(* PLC project Система умного дома.project, CODESYS CODESYS V3.5 SP17 Patch 3 *)
(* stored: creationDateTime 2026-04-06T20:38:17.5908527, modificationDateTime 2026-03-25T09:46:39.3897592 *)

{attribute 'qualified_only'}
{attribute 'strict'}
TYPE E_ALERT_PRIORITY : (ALERT_PRIORITY_NONE := 0, ALERT_PRIORITY_LOW := 1, ALERT_PRIORITY_MEDIUM := 2, ALERT_PRIORITY_HIGH := 3, ALERT_PRIORITY_CRITICAL := 4) BYTE;
END_TYPE

{attribute 'qualified_only'}
{attribute 'strict'}
TYPE E_Debug_Log_Level : (LOG_LEVEL_MINIMAL := 0, LOG_LEVEL_NORMAL := 1, LOG_LEVEL_VERBOSE := 2, LOG_LEVEL_DEBUG := 3) BYTE;
END_TYPE

{attribute 'qualified_only'}
{attribute 'strict'}
TYPE E_Lifetime_Device_Type : (LIFETIME_DEVICE_PUMP := 1, LIFETIME_DEVICE_FAN := 2) BYTE;
END_TYPE

{attribute 'qualified_only'}
{attribute 'strict'}
TYPE E_Outdoor_Mode : (OUTDOOR_MODE_AUTO := 0, OUTDOOR_MODE_PARTY := 1, OUTDOOR_MODE_SECURITY := 2, OUTDOOR_MODE_ECONOMY := 3, OUTDOOR_MODE_MANUAL := 4) BYTE;
END_TYPE

{attribute 'qualified_only'}
{attribute 'strict'}
TYPE E_PLC_ROLE : (ROLE_UNDEFINED := 0, ROLE_ACTIVE := 1, ROLE_STANDBY := 2, ROLE_OFFLINE := 3) USINT;
END_TYPE

{attribute 'qualified_only'}
{attribute 'strict'}
TYPE E_Rule_Action_Type : (ACTION_NONE := 0, ACTION_SET_FLOOR_HEATING := 1, ACTION_SET_LIGHTING_BASE := 2, ACTION_SET_LIGHTING_ACCENT := 3, ACTION_SET_SOCKET := 4, ACTION_SET_VENTILATION := 5, ACTION_SET_BLINDS := 6, ACTION_ACTIVATE_SCENARIO := 7, ACTION_TOGGLE_LIGHTING := 8, ACTION_TOGGLE_SOCKET := 9) BYTE;
END_TYPE

{attribute 'qualified_only'}
{attribute 'strict'}
TYPE E_Rule_Comparison : (COMP_NONE := 0, COMP_EQ := 1, COMP_GT := 2, COMP_LT := 3, COMP_GE := 4, COMP_LE := 5, COMP_IN_RANGE := 6, COMP_TRUE := 7, COMP_FALSE := 8) BYTE;
END_TYPE

(* values of E_Rule_Condition_Type: COND_AND: Логическое И (Rule Chaining); COND_OR: Логическое ИЛИ (Rule Chaining) *)

{attribute 'qualified_only'}
{attribute 'strict'}
TYPE E_Rule_Condition_Type : (COND_NONE := 0, COND_AIR_TEMP := 1, COND_FLOOR_TEMP := 2, COND_HUMIDITY := 3, COND_CO2 := 4, COND_METHANE := 5, COND_CO := 6, COND_DOOR_WINDOW := 7, COND_FLOOD := 8, COND_SMOKE := 9, COND_MOTION := 10, COND_TIME_OF_DAY := 11, COND_DAY_OF_WEEK := 12, COND_AND := 13, COND_OR := 14) BYTE;
END_TYPE

{attribute 'qualified_only'}
{attribute 'strict'}
TYPE E_SCENARIO_TYPE : (SCENARIO_NONE := 0, SCENARIO_MORNING := 1, SCENARIO_EVENING := 2, SCENARIO_AWAY := 3, SCENARIO_PARTY := 4, SCENARIO_SLEEP := 5, SCENARIO_EMERGENCY := 6, SCENARIO_PRESENCE := 7) BYTE;
END_TYPE

{attribute 'qualified_only'}
{attribute 'strict'}
TYPE E_SENSOR_TYPE : (SENSOR_TYPE_NONE := 0, SENSOR_TYPE_DOOR_WINDOW := 5, SENSOR_TYPE_GLASS_BREAK := 6, SENSOR_TYPE_FLOOD := 7, SENSOR_TYPE_SMOKE := 8, SENSOR_TYPE_GAS_METHANE := 1, SENSOR_TYPE_GAS_CO := 2, SENSOR_TYPE_TEMP_FLOOR := 3, SENSOR_TYPE_TEMP_AIR := 4) USINT;
END_TYPE

{attribute 'qualified_only'}
{attribute 'strict'}
TYPE E_Trend_Parameter_Type : (TREND_PARAM_NONE := 0, TREND_PARAM_TEMP_AIR := 1, TREND_PARAM_TEMP_FLOOR := 2, TREND_PARAM_PRESSURE := 3, TREND_PARAM_PUMP_CURRENT := 4, TREND_PARAM_GAS_METHANE := 5, TREND_PARAM_GAS_CO := 6) BYTE;
END_TYPE

{attribute 'qualified_only'}
{attribute 'strict'}
TYPE E_TwoFactor_Method : (TF_METHOD_NONE := 0, TF_METHOD_RFID := 1, TF_METHOD_TOTP := 2, TF_METHOD_BOTH := 3) BYTE;
END_TYPE

{attribute 'qualified_only'}
{attribute 'strict'}
TYPE E_Valve_Test_Result : (TEST_RESULT_NONE := 0, TEST_RESULT_PASSED := 1, TEST_RESULT_CURRENT_DEVIATION := 2, TEST_RESULT_TIME_DEVIATION := 3, TEST_RESULT_STALL := 4, TEST_RESULT_LIMIT_SWITCH_FAIL := 5, TEST_RESULT_ABORTED := 6) BYTE;
END_TYPE

(* values of E_VALVE_TYPE: VALVE_NC: Нормально-закрытый; VALVE_NO: Нормально-открытый *)

{attribute 'qualified_only'}
{attribute 'strict'}
TYPE E_VALVE_TYPE : (VALVE_NC := 1, VALVE_NO := 2) USINT;
END_TYPE

{attribute 'qualified_only'}
{attribute 'strict'}
TYPE E_VENTILATION_LOCATION : (VENT_LOCATION_NONE := 0, VENT_LOCATION_BASEMENT_GAME_ROOM := 1, VENT_LOCATION_BASEMENT_GYM := 2, VENT_LOCATION_BASEMENT_BOILER_ROOM := 3, VENT_LOCATION_BATHROOM_1F := 4, VENT_LOCATION_BATHROOM_2F := 5, VENT_LOCATION_MASTER_BATHROOM := 6, VENT_LOCATION_LAUNDRY := 7, VENT_LOCATION_KITCHEN := 8) BYTE;
END_TYPE

{attribute 'qualified_only'}
{attribute 'strict'}
TYPE E_VENTILATION_UNIT_TYPE : (VENTILATION_TYPE_NONE := 0, VENTILATION_TYPE_SUPPLY := 1, VENTILATION_TYPE_EXHAUST := 2) USINT;
END_TYPE

{attribute 'qualified_only'}
{attribute 'strict'}
TYPE E_WEATHER_COMPENSATION_METHOD : (WEATHER_COMP_NONE := 0, WEATHER_COMP_OUTDOOR_RESET := 1) USINT;
END_TYPE

{attribute 'qualified_only'}
{attribute 'strict'}
TYPE E_Zone_Access_Level : (ZONE_ACCESS_NONE := 0, ZONE_ACCESS_VIEW := 1, ZONE_ACCESS_CONTROL := 2, ZONE_ACCESS_CONFIG := 3, ZONE_ACCESS_FULL := 4) BYTE;
END_TYPE

TYPE ST_Astro_Time : STRUCT
  sunrise_ms : UDINT := 0;
  sunset_ms : UDINT := 0;
  is_daylight : BOOL := FALSE;
END_STRUCT;
END_TYPE

TYPE ST_BlackBox_Record : STRUCT
  Timestamp : UDINT;
  Gas_Methane_LEL : REAL;
  Gas_CO_PPM : REAL;
  Flood_Active : BOOL;
  Fire_Active : BOOL;
  Valve_Gas_Status : BYTE;
  Valve_Water_Status : BYTE;
  PLC_Active_ID : BYTE;
END_STRUCT;
END_TYPE

TYPE ST_Boiler_Status : STRUCT
  Active : BOOL;
  Running : BOOL;
  Error : BOOL;
  Power_Percent : REAL;
  Current_Power : REAL;
  Work_Seconds : UDINT;
  Work_Hours : REAL;
  Resource_Percent : REAL := 100;
  Last_Start : DT;
END_STRUCT;
END_TYPE

TYPE ST_Component_Maintenance : STRUCT
  Is_Faulty : BOOL;  (* Устройство неисправно *)
  Is_In_Maintenance : BOOL;  (* Выведено в ремонт вручную *)
  Fallback_Value : REAL;  (* Значение для подстановки (0-100% или температура) *)
  Use_Last_Good_Value : BOOL;  (* Использовать последнее достоверное значение *)
END_STRUCT;
END_TYPE

TYPE ST_Debug_Log_Record : STRUCT
  timestamp_ms : UDINT;
  level : BYTE;  (* E_Debug_Log_Level *)
  source_id : BYTE;
  event_code : WORD;
  value_int : UDINT;
  value_real : REAL;
  text : STRING(80);
  crc32 : DWORD;
END_STRUCT;
END_TYPE

TYPE ST_Debug_Logger_Config : STRUCT
  enabled : BOOL;
  sampling_period_ms : UDINT := 1000;
END_STRUCT;
END_TYPE

TYPE ST_Device_Health : STRUCT
  Health_Score : BYTE := 100;  (* 0..100% *)
  Total_Runtime_Hours : UDINT;
  Starts_Count : UDINT;
  Last_Start_Current : REAL;
  Avg_Start_Current : REAL;
  Maintenance_Required : BOOL;
  Warning_Message : STRING(50);
END_STRUCT;
END_TYPE

TYPE ST_DHW_Config : STRUCT
  Target_Temp : REAL := 55;
  Hysteresis : REAL := 2;
  Circulation_Schedule_Enabled : BOOL := TRUE;
  Circulation_Start : TOD := TIME_OF_DAY#6:0;
  Circulation_End : TOD := TIME_OF_DAY#23:0;
  Anti_Legionella_Enabled : BOOL := TRUE;
  Anti_Legionella_Day : UINT := 7;  (* Воскресенье *)
END_STRUCT;
END_TYPE

TYPE ST_DHW_Status : STRUCT
  Temp : REAL;
  Pressure : REAL;
  Heating_Pump_On : BOOL;
  Circ_Pump_On : BOOL;
  Error : BOOL;
  Error_ID : WORD;
END_STRUCT;
END_TYPE

TYPE ST_Flood_Config : STRUCT
  Emergency_Two_Stage_Enabled : BOOL := TRUE;  (* ТЗ 4.4 *)
  Valve_Test_Period_Days : UINT := 7;  (* ТЗ 12.2 *)
  Current_Threshold_MA : REAL := 500;  (* Порог тока для диагностики *)
END_STRUCT;
END_TYPE

TYPE ST_Flood_Global_Config : STRUCT
  valve_types : ARRAY[1..3] OF E_VALVE_TYPE := [3(E_VALVE_TYPE.VALVE_NC)];
  min_duration_ms : UDINT := 30000;
END_STRUCT;
END_TYPE

TYPE ST_FloorHeating_Circuit_Config : STRUCT
  circuit_id : BYTE := 0;
  zone : BYTE := 0;
  design_temp : REAL := 35;
  min_temp : REAL := 20;
  max_temp : REAL := 45;
  pid_kp : REAL := 2;
END_STRUCT;
END_TYPE

TYPE ST_FloorHeating_Global_Config : STRUCT
  enable_floor_heating : BOOL := TRUE;
  anti_freeze_temp : REAL := 7;
  overheat_temp : REAL := 45;
  weather_compensation_enabled : BOOL := TRUE;
  total_circuits : BYTE := 16;
END_STRUCT;
END_TYPE

TYPE ST_FloorHeating_Manifold_Config : STRUCT
  manifold_id : BYTE;
  location : STRING(30);
  nominal_flow : REAL;
  enable_pump : BOOL;
  circuits : ARRAY[1..4] OF ST_FloorHeating_Circuit_Config;
END_STRUCT;
END_TYPE

TYPE ST_Gas_Valve_Configuration : STRUCT
  valve_id : BYTE := 0;
  valve_type : E_VALVE_TYPE := E_VALVE_TYPE.VALVE_NC;
  close_time_seconds : UDINT := 10;
  open_time_seconds : UDINT := 10;
  emergency_open_allowed : BOOL := FALSE;
END_STRUCT;
END_TYPE

TYPE ST_Gateway_Command : STRUCT
  command_id : UDINT;
  timestamp_ms : UDINT;
  operator_id : STRING(10);
  command_type : BYTE;
  target_zone : BYTE;
  target_value : REAL;
  target_on_off : BOOL;
  target_scenario : E_SCENARIO_TYPE;
  target_armed : BOOL;
  crc32 : DWORD;
END_STRUCT;
END_TYPE

TYPE ST_Heating_Config : STRUCT
  Weather_Comp_Enabled : BOOL := TRUE;
  Weather_Coef : REAL := 0.1;
  Freeze_Threshold : REAL := 7;
  Overheat_Threshold : REAL := 45;
  Night_Reduction : REAL := 3;
  Target_Floor_Temp : REAL := 28;
  Target_Room_Temp : REAL := 22;
  Hysteresis : REAL := 0.5;
END_STRUCT;
END_TYPE

TYPE ST_History_Record : STRUCT
  timestamp_ms : UDINT := 0;
  event_code : WORD := 0;
  event_value : REAL := 0;
  unit : BYTE := 0;
  zone_id : BYTE := 0;
  operator_id : STRING(10) := '';
  priority : E_ALERT_PRIORITY := E_ALERT_PRIORITY.ALERT_PRIORITY_NONE;
END_STRUCT;
END_TYPE

TYPE ST_Lifetime_Status : STRUCT
  device_id : BYTE;
  runtime_hours : UDINT;
  start_count : UDINT;
  remaining_hours : UDINT;
  remaining_percent : BYTE;
  maintenance_required : BOOL;
  last_calc_timestamp : UDINT;
END_STRUCT;
END_TYPE

TYPE ST_Maintenance_Access_Config : STRUCT
  maintenance_enabled : BOOL := FALSE;
  max_duration_minutes : UDINT := 60;
  requires_two_person : BOOL := TRUE;
  access_level_required : BYTE := 2;
END_STRUCT;
END_TYPE

TYPE ST_Manifold_Status : STRUCT
  Pump_On : BOOL;
  Pump_Current : REAL;
  Pressure : REAL;
  Temp_Supply : REAL;
  Temp_Return : REAL;
  Valve_Pos : REAL;  (* 0-100% *)
  Error : BOOL;
  Error_ID : WORD;
END_STRUCT;
END_TYPE

TYPE ST_Operator_Zone_Rights : STRUCT
  operator_id : STRING(10);
  global_access_level : BYTE := 0;
  zone_masks : ARRAY[1..18] OF DWORD;
  last_modified : UDINT;
END_STRUCT;
END_TYPE

TYPE ST_Outdoor_Zone_Config : STRUCT
  zone_id : BYTE := 0;
  lighting_circuit_id : BYTE := 0;
  auto_enabled : BOOL := TRUE;
  party_mode_enabled : BOOL := FALSE;
END_STRUCT;
END_TYPE

TYPE ST_Owen_Analog_Value : STRUCT
  rValue : REAL;  (* Измеренное значение *)
  uiCycleTime : UINT;  (* Циклическое время *)
  wStatus : WORD;  (* Код статуса (ANALOG_SENSOR_ERRORS) *)
END_STRUCT;
END_TYPE

TYPE ST_Rule_Action : STRUCT
  Active : BOOL;
  Target_ID : BYTE;
  Value : REAL;
END_STRUCT;
END_TYPE

TYPE ST_Scenario_Config : STRUCT
  scenario_id : E_SCENARIO_TYPE;
  lighting_level_base : BYTE := 100;
  lighting_level_accent : BYTE := 100;
  floor_heating_adjust_celsius : REAL := 0;
  ventilation_speed_percent : BYTE := 50;
  sockets_enabled : BOOL := TRUE;
  blinds_position_percent : BYTE := 0;
END_STRUCT;
END_TYPE

TYPE ST_Scenario_Transition_Config : STRUCT
  current_scenario : E_SCENARIO_TYPE;
  target_scenario : E_SCENARIO_TYPE;
  min_duration_minutes : UDINT := 5;
  transition_allowed : BOOL := FALSE;
END_STRUCT;
END_TYPE

TYPE ST_Security_Config : STRUCT
  PIN_Code : STRING(4) := '1234';
  Max_Attempts : UINT := 3;
  Entry_Delay_S : UINT := 45;
  Two_Factor_Enabled : BOOL := FALSE;
  Two_Stage_Mode : BOOL := TRUE;  (* ТЗ 3.4 *)
  Confirmation_Timeout_S : UINT := 120;  (* ТЗ 3.4 (60-300с) *)
  Phones : ARRAY[1..5] OF STRING(15);
  gate_open_pulse_ms : UDINT := 1000;  (* Управление доступом *)
  wicket_open_pulse_ms : UDINT := 1000;
  lock_open_pulse_ms : UDINT := 1000;
  lock_close_pulse_ms : UDINT := 1000;
END_STRUCT;
END_TYPE

TYPE ST_Security_Global_Config : STRUCT
  entry_delay_seconds : UDINT := 30;
  exit_delay_seconds : UDINT := 60;
  alarm_duration_seconds : UDINT := 180;
  two_person_timeout_seconds : UDINT := 120;
  max_access_attempts : BYTE := 3;
  auto_arm_enabled : BOOL := FALSE;
  auto_arm_time_ms : UDINT := 0;
  gate_open_pulse_ms : UDINT := 1000;  (* ТЗ: Управление доступом *)
  wicket_open_pulse_ms : UDINT := 1000;
  lock_open_pulse_ms : UDINT := 1000;
  lock_close_pulse_ms : UDINT := 1000;
END_STRUCT;
END_TYPE

TYPE ST_Security_Zone_State : STRUCT
  Armed : BOOL;
  Alarm : BOOL;
  Bypassed : BOOL;
  Last_Trigger_Time : DT;
  Trigger_Count : UINT;
END_STRUCT;
END_TYPE

TYPE ST_Sensor_Calibration_Record : STRUCT
  sensor_id : UDINT := 0;
  sensor_type : E_SENSOR_TYPE;
  zone_id : BYTE := 0;
  offset : REAL := 0;
  multiplier : REAL := 1;
  last_calibration_timestamp : UDINT := 0;
  verification_passed : BOOL := FALSE;
END_STRUCT;
END_TYPE

TYPE ST_State_Snapshot : STRUCT
  timestamp_ms : UDINT := 0;
  operator_id : STRING(10) := '';
  scenario_id : E_SCENARIO_TYPE := E_SCENARIO_TYPE.SCENARIO_NONE;
  lighting_levels : ARRAY[1..16] OF BYTE;
  floor_heating_setpoints : ARRAY[1..16] OF REAL;
  alarm_active : BOOL := FALSE;
  crc32 : DWORD := 0;
END_STRUCT;
END_TYPE

TYPE ST_System_State_Summary : STRUCT
  Outdoor_Temp : REAL;
  Indoor_Temp : ARRAY[1..16] OF REAL;
  Floor_Temps : ARRAY[1..16] OF REAL;
  Humidity : ARRAY[1..8] OF REAL;
  CO2 : ARRAY[1..8] OF REAL;
  Gas_Alarm : BOOL;
  Flood_Alarm : BOOL;
  Fire_Alarm : BOOL;
  Security_Armed : BOOL;
END_STRUCT;
END_TYPE

TYPE ST_Tariff_Config : STRUCT
  Enabled : BOOL := FALSE;
  Night_Start_Hour : UINT := 23;  (* 23:00 *)
  Night_End_Hour : UINT := 7;  (* 07:00 *)
  Boost_Delta : REAL := 2;  (* На сколько градусов поднять уставку ночью *)
END_STRUCT;
END_TYPE

TYPE ST_Trend_Config : STRUCT
  param_type : BYTE;  (* E_Trend_Parameter_Type *)
  zone_id : BYTE;
  enabled : BOOL;
  deviation_threshold_percent : REAL := 10;
  history_days : UDINT := 7;
END_STRUCT;
END_TYPE

TYPE ST_Trend_Data : STRUCT
  config : ST_Trend_Config;
  record_count : UDINT;
  write_index : UDINT;
  sum_values : REAL;
  crc32 : DWORD;
END_STRUCT;
END_TYPE

TYPE ST_Trend_Header : STRUCT
  parameter_type : BYTE;  (* E_Trend_Parameter_Type *)
  zone_id : BYTE := 0;
  records_count : UDINT := 0;
  average_value : REAL := 0;
  min_value : REAL := 0;
  max_value : REAL := 0;
END_STRUCT;
END_TYPE

TYPE ST_Trend_History_Record : STRUCT
  timestamp_ms : UDINT := 0;
  value : REAL := 0;
END_STRUCT;
END_TYPE

TYPE ST_TwoFactor_Auth_State : STRUCT
  operator_id : STRING(10);
  is_pending : BOOL;  (* Ожидание ввода 2-го фактора *)
  start_time : UDINT;
  timeout_ms : UDINT := 60000;
END_STRUCT;
END_TYPE

TYPE ST_TwoFactor_Data : STRUCT
  operator_id : STRING(10);
  AuthMethod : BYTE;  (* E_TwoFactor_Method *)
  rfid_tag : STRING(20);
  totp_secret : STRING(32);
  last_modified : UDINT;
END_STRUCT;
END_TYPE

TYPE ST_User_Rule : STRUCT
  Enabled : BOOL;
  Condition_Type : BYTE;  (* 1-Temp, 2-Hum, 3-CO2, 4-Security, 5-Time *)
  Condition_Op : BYTE;  (* 1:>, 2:<, 3:= *)
  Condition_Value : REAL;
  Action_Target_ID : BYTE;
  Action_Value : REAL;
  Action_Type : BYTE;  (* 1-SetTemp, 2-Switch, 3-Scenario *)
  Priority : BYTE;  (* ТЗ 7.4: Приоритет (0-255) *)
END_STRUCT;
END_TYPE

TYPE ST_Valve_Test_Config : STRUCT
  valve_id : BYTE := 0;
  test_interval_days : UDINT := 7;
  nominal_current_a : REAL := 0.5;
  Nominal_Current : REAL := 0.5;
  nominal_close_time_sec : REAL := 10;
  enabled : BOOL := TRUE;
END_STRUCT;
END_TYPE

TYPE ST_Ventilation_Config : STRUCT
  CO2_Threshold : REAL := 800;
  Humidity_Threshold : REAL := 65;
  Night_Mode_Start : TOD := TIME_OF_DAY#23:0;
  Night_Mode_End : TOD := TIME_OF_DAY#7:0;
END_STRUCT;
END_TYPE

TYPE ST_Ventilation_Global_Config : STRUCT
  enable_ventilation : BOOL := TRUE;
  total_units : BYTE := 8;
  default_supply_speed : BYTE := 40;
  default_exhaust_speed : BYTE := 40;
END_STRUCT;
END_TYPE

TYPE ST_Ventilation_Scenario_Mode : STRUCT
  Scenario_ID : BYTE;
  Scenario_Priority : BYTE;
  Fire_Alarm : BOOL;
  Methane_Alarm : BOOL;
  Smoke_Detected : BOOL;
  Exhaust_Modes : ARRAY[1..5] OF BYTE;
  Supply_Modes : ARRAY[1..3] OF BYTE;
END_STRUCT;
END_TYPE

TYPE ST_Ventilation_Unit : STRUCT
  Enabled : BOOL;
  Speed_Percent : REAL;
  Filter_Dirty : BOOL;
  Error : BOOL;
  Mode : BYTE;  (* 0-Eco, 1-Std, 2-Int, 3-Emergency *)
END_STRUCT;
END_TYPE

TYPE ST_Ventilation_Unit_Config : STRUCT
  unit_id : BYTE := 0;
  unit_type : E_VENTILATION_UNIT_TYPE;
  location : E_VENTILATION_LOCATION;
  min_speed : BYTE := 20;
  max_speed : BYTE := 100;
  Threshold_Hum : REAL := 65;
  has_smoke_detector : BOOL := FALSE;
END_STRUCT;
END_TYPE

TYPE ST_Zone_Sensors : STRUCT
  Temp_Room : REAL;
  Temp_Floor : REAL;
  Motion_Active : BOOL;
  Switch_Physical : BOOL;
  Light_State : BOOL;
  Maintenance : ST_Component_Maintenance;
END_STRUCT;
END_TYPE

{attribute 'qualified_only'}
VAR_GLOBAL  (* GVL_BlackBox *)
  G_BlackBox_Buffer : ARRAY[0..99] OF ST_BlackBox_Record;  (* Буфер на 100 записей (при опросе 100мс это 10 секунд истории) *)
  G_BlackBox_Frozen : BOOL;
  G_BlackBox_LastIndex : INT;
END_VAR

{attribute 'qualified_only'}
VAR_GLOBAL CONSTANT  (* GVL_Constants *)
  C_MS_PER_SEC : UDINT := 1000;
  C_SEC_PER_MIN : UDINT := 60;
  C_MIN_PER_HOUR : UDINT := 60;
  C_MS_PER_MIN : UDINT := 60000;
  C_MAX_RULES : INT := 20;
  C_ZONE_COUNT : BYTE := 18;
END_VAR

{attribute 'qualified_only'}
VAR_GLOBAL  (* GVL_Diagnostics *)
  G_Pump_Health : ARRAY[1..5] OF ST_Device_Health;  (* Для 5 коллекторных насосов *)
  G_Gas_Valve_Health : ST_Device_Health;
  G_System_Health_Summary : BYTE := 100;
END_VAR

{attribute 'qualified_only'}
VAR_GLOBAL  (* GVL_Global_Variables *)
  GVL_System_Time_MS : UDINT;
  GVL_IsActivePLC : BOOL := TRUE;
  GVL_Local_PLC_Role : E_PLC_ROLE := E_PLC_ROLE.ROLE_ACTIVE;
  GVL_Floor_Temps : ARRAY[1..16] OF REAL;  (* Данные датчиков *)
  GVL_Valve_States : ARRAY[1..3] OF BYTE;
END_VAR

VAR_GLOBAL  (* GVL_HMI_Config *)
  G_HMI_FloorHeating_Configs : ARRAY[1..16] OF ST_FloorHeating_Circuit_Config;  (* Настройки отопления (16 контуров) *)
  G_HMI_Tariff_Settings : ST_Tariff_Config;
  G_HMI_Vent_Global_Config : ST_Ventilation_Global_Config;  (* Настройки вентиляции (8 установок) *)
  G_HMI_Vent_Unit_Configs : ARRAY[1..8] OF ST_Ventilation_Unit_Config;
  G_HMI_Scenario_Configs : ARRAY[1..6] OF ST_Scenario_Config;  (* Для каждого типа сценария *)
  G_HMI_Outdoor_Configs : ARRAY[1..4] OF ST_Outdoor_Zone_Config;
  G_HMI_Flood_Config : ST_Flood_Global_Config;  (* Настройки безопасности *)
  G_HMI_Cleaning_Mode_Active : ARRAY[1..3] OF BOOL;  (* Режим уборки для 3-х зон протечки *)
  G_HMI_Cleaning_Mode_TimeLeft : ARRAY[1..3] OF UINT;  (* Оставшееся время (мин) *)
  G_HMI_Gas_Config : ST_Gas_Valve_Configuration;
  G_HMI_Admin_2FA_Enabled : BOOL := FALSE;  (* Настройка: 1 или 2 фактора для ADMIN *)
  G_HMI_Current_Operator_Factor2_Done : BOOL;  (* Флаг прохождения 2-го фактора *)
  G_HMI_Sensor_Calibrations : ARRAY[1..20] OF ST_Sensor_Calibration_Record;  (* Калибровка датчиков (например, для 20 датчиков) *)
  G_HMI_Current_Operator_ID : STRING(10);  (* ID текущего авторизованного пользователя *)
  G_HMI_Manual_Gas_Valve_Open : BOOL;  (* Запрос на открытие *)
  G_HMI_Manual_Gas_Valve_Time : UDINT := 5;  (* Время в минутах *)
  G_HMI_Manual_Gas_Valve_TimeLeft : UDINT;  (* Оставшееся время (для вывода на HMI) *)
  G_HMI_Apply_Settings : BOOL;  (* Команда на сохранение настроек в NVRAM *)
  G_HMI_Gate_Open_Req : BOOL;  (* Управление доступом (HMI) *)
  G_HMI_Wicket_Open_Req : BOOL;
  G_HMI_Lock_1_Open_Req : BOOL;
  G_HMI_Lock_1_Close_Req : BOOL;
  G_HMI_Lock_2_Open_Req : BOOL;
  G_HMI_Lock_2_Close_Req : BOOL;
END_VAR

VAR_GLOBAL  (* GVL_IO *)
  DI_Security_Open : ARRAY[1..15] OF BOOL;  (* Датчики открытия (15 физических каналов по ТЗ 3.1) *)
  DI_Security_Glass : ARRAY[1..15] OF BOOL;  (* Датчики разбития (15 физических каналов по ТЗ 3.2) *)
  DI_Security_2F_Group : BOOL;  (* Групповой канал 2-го этажа *)
  DI_Flood_Sensors : ARRAY[1..12] OF BOOL;  (* Датчики протечки (12 штук по ТЗ 4.1) *)
  AO_Manifold_Valves : ARRAY[1..5] OF UINT;  (* 0-1000 (Modbus) *)
  DO_Manifold_Pumps : ARRAY[1..5] OF BOOL;
  AI_Manifold_Currents : ARRAY[1..5] OF INT;  (* 4-20mA -> 400-2000 *)
  AI_Manifold_Pressures : ARRAY[1..5] OF INT;  (* 0-10V -> 0-1000 *)
  AI_Manifold_Temps_Supply : ARRAY[1..5] OF ST_Owen_Analog_Value;
  AI_Manifold_Temps_Return : ARRAY[1..5] OF INT;
  AO_Supply_Fans : ARRAY[1..3] OF UINT;  (* 0-1000 *)
  AO_Exhaust_Fans : ARRAY[1..5] OF UINT;  (* 0-1000 *)
  DO_Boiler_Enable : ARRAY[1..2] OF BOOL;  (* Котлы (BAXI Luna Platinum+ через OpenTherm) *)
  AO_Boiler_Setpoint : ARRAY[1..2] OF UINT;  (* 0-1000 (0-100.0 C) *)
  AI_Boiler_Modulation : ARRAY[1..2] OF INT;
  AI_Boiler_Flame_Status : ARRAY[1..2] OF BOOL;
  DI_Boiler_Error : ARRAY[1..2] OF BOOL;
  AI_Methane_LEL : ARRAY[1..2] OF ST_Owen_Analog_Value;  (* 0-100% LEL *)
  AI_CO_PPM : ARRAY[1..8] OF REAL;  (* 0-1000 PPM *)
  DI_Smoke_Sensors : ARRAY[1..6] OF BOOL;
  AI_Temp_Outdoor : ST_Owen_Analog_Value;  (* Аналоговые входы (AI) *)
  AI_Floor_Temps : ARRAY[1..16] OF REAL;
  AI_Room_Temps : ARRAY[1..16] OF REAL;  (* Датчики температуры помещения (ТЗ 1.1) *)
  DO_Zone_Valves : ARRAY[1..16] OF BOOL;  (* Клапаны контуров ТП *)
  AI_DHW_Temp : REAL;  (* ГВС (ТЗ 5.0) *)
  AI_DHW_Pressure : REAL;
  DO_DHW_Heating_Pump : BOOL;
  DO_DHW_Circ_Pump : BOOL;
  DI_Lighting_Switches : ARRAY[1..16] OF BOOL;  (* Освещение и Движение (ТЗ 1.0, 2.0) *)
  DI_Motion_Sensors : ARRAY[1..16] OF BOOL;
  DO_Gas_Valve_Close : BOOL;  (* Безопасность и Аварии *)
  DO_Water_Valve_35_Close : BOOL;
  DO_Water_Valve_36_Close : BOOL;
  AI_Water_Valve_35_Current : REAL;
  AI_Water_Valve_36_Current : REAL;
  DI_Power_OK : BOOL;
  DO_Gas_Siren : BOOL;
  DO_Fire_Siren : BOOL;
  DO_Pump_Main_Enable : BOOL;
  DO_Gate_Open : BOOL;  (* Управление доступом (Сухие контакты) *)
  DO_Wicket_Open : BOOL;
  DO_Lock_1_Open : BOOL;
  DO_Lock_1_Close : BOOL;
  DO_Lock_2_Open : BOOL;
  DO_Lock_2_Close : BOOL;
END_VAR

VAR_GLOBAL  (* GVL_Vars *)
  G_System_Time_MS : UDINT;  (* Системное время (мс) *)
  G_Current_Scenario : E_SCENARIO_TYPE := E_SCENARIO_TYPE.SCENARIO_NONE;
  G_Security_Armed : BOOL := FALSE;
  G_Gas_Alarm_Active : BOOL := FALSE;
  G_Fire_Alarm_Active : BOOL := FALSE;
  G_Flood_Alarm_Active : BOOL := FALSE;
  G_Local_PLC_ID : BYTE := 1;  (* ID текущего ПЛК (1 для A, 2 для B) *)
  G_Active_PLC_ID : BYTE := 1;  (* ID активного ПЛК в данный момент *)
  G_Remote_PLC_Pulse : BOOL;  (* Импульс от партнера *)
  G_HMI_Current_Operator_ID : STRING(10) := 'ADMIN';  (* HMI и Конфигурация *)
  G_HMI_Gas_Config : ST_Gas_Valve_Configuration;
  G_Heating_Config : ST_Heating_Config;
  G_Ventilation_Config : ST_Ventilation_Config;
  G_DHW_Config : ST_DHW_Config;
  G_Security_Config : ST_Security_Config;
  G_Flood_Config : ST_Flood_Config;
  G_HMI_Mute_Alarm : BOOL;
  G_HMI_Manual_Gas_Valve_Open : BOOL;
  G_HMI_Manual_Gas_Valve_Time : UDINT := 300000;  (* 5 минут по умолчанию *)
  G_HMI_Manual_Gas_Valve_TimeLeft : UDINT;
  G_Floor_Temps : ARRAY[1..16] OF REAL;  (* Состояние датчиков *)
  G_BlackBox_Buffer : ARRAY[0..99] OF ST_BlackBox_Record;  (* Черный ящик *)
  G_BlackBox_LastIndex : INT;
  G_BlackBox_Frozen : BOOL;
  G_Maintenance_Zones : ARRAY[1..16] OF ST_Component_Maintenance;  (* ТЗ 6.0: Обслуживание и ремонт *)
  G_Maintenance_Manifolds : ARRAY[1..5] OF ST_Component_Maintenance;
  G_Maintenance_Lighting : ARRAY[1..16] OF ST_Component_Maintenance;
  G_HMI_Gate_Open_Req : BOOL;  (* Управление доступом (HMI) *)
  G_HMI_Wicket_Open_Req : BOOL;
  G_HMI_Lock_1_Open_Req : BOOL;
  G_HMI_Lock_1_Close_Req : BOOL;
  G_HMI_Lock_2_Open_Req : BOOL;
  G_HMI_Lock_2_Close_Req : BOOL;
END_VAR

INTERFACE IValveController
METHOD OpenValve : BOOL
  VAR_INPUT
    VI_Operator_ID : STRING(10);
    VI_Force : BOOL;
  END_VAR
END_METHOD
METHOD CloseValve : BOOL
  VAR_INPUT
    VI_Operator_ID : STRING(10);
    VI_Force : BOOL;
  END_VAR
END_METHOD
METHOD GetStatus : BYTE
END_METHOD
END_INTERFACE

FUNCTION_BLOCK FB_AccessCode_Manager
  VAR_INPUT
    VI_System_Time_MS : UDINT;
    VI_IsActivePLC : BOOL;
    VI_Code_To_Check : STRING(4);
    VI_RFID_To_Check : STRING(20);
  END_VAR
  VAR_OUTPUT
    VO_Code_Valid : BOOL;
  END_VAR
  VAR_IN_OUT
    VI_Access_Codes : ARRAY[1..GVL_CONSTANTS.C_MAX_ACCESS_CODES] OF DWORD;
    VI_RFID_Tags : ARRAY[1..GVL_CONSTANTS.C_MAX_ACCESS_CODES] OF STRING(20);
  END_VAR
  VAR
    L_i : INT;
    pCode : POINTER TO BYTE;
    L_CRC_Calc : FB_CRC32_Calculator;
    L_Input_Hash : DWORD;
  END_VAR

            VO_Code_Valid := FALSE;

// Вычисляем хэш введенного кода
IF LEN(VI_Code_To_Check) > 0 THEN
    pCode := ADR(VI_Code_To_Check);
    L_Input_Hash := 0;
    FOR L_i := 1 TO GVL_CONSTANTS.C_MAX_ACCESS_CODES DO
        IF VI_Access_Codes[L_i] <> 0 AND VI_Access_Codes[L_i] = L_Input_Hash THEN
            VO_Code_Valid := TRUE;
            RETURN;
        END_IF;
    END_FOR;
END_IF;

// Проверяем RFID метку
IF LEN(VI_RFID_To_Check) > 0 THEN
    FOR L_i := 1 TO GVL_CONSTANTS.C_MAX_ACCESS_CODES DO
        IF VI_RFID_Tags[L_i] <> '' AND VI_RFID_Tags[L_i] = VI_RFID_To_Check THEN
            VO_Code_Valid := TRUE;
            RETURN;
        END_IF;
    END_FOR;
END_IF;
// >>> BULK_SYNC_ANCHOR: FB_AccessCode_Manager <<<
          
END_FUNCTION_BLOCK

FUNCTION_BLOCK FB_Access_Control
  VAR_INPUT
    VI_System_Time_MS : UDINT;
    VI_IsActivePLC : BOOL;
    VI_Armed : BOOL;
    VI_System_Mode : E_System_Operating_Mode;
    VI_Gate_Open_Req : BOOL;
    VI_Wicket_Open_Req : BOOL;
    VI_Lock_1_Open_Req : BOOL;
    VI_Lock_1_Close_Req : BOOL;
    VI_Lock_2_Open_Req : BOOL;
    VI_Lock_2_Close_Req : BOOL;
    VI_PIN_Code : STRING(4);
    VI_RFID_Tag : STRING(20);
    VI_Config : ST_Security_Global_Config;
  END_VAR
  VAR_OUTPUT
    VO_Gate_Open : BOOL;
    VO_Wicket_Open : BOOL;
    VO_Lock_1_Open : BOOL;
    VO_Lock_1_Close : BOOL;
    VO_Lock_2_Open : BOOL;
    VO_Lock_2_Close : BOOL;
  END_VAR
  VAR_IN_OUT
    VI_Access_Codes : ARRAY[1..GVL_CONSTANTS.C_MAX_ACCESS_CODES] OF DWORD;
    VI_RFID_Tags : ARRAY[1..GVL_CONSTANTS.C_MAX_ACCESS_CODES] OF STRING(20);
  END_VAR
  VAR
    L_Gate_Timer : TP;
    L_Wicket_Timer : TP;
    L_Lock_1_Open_T : TP;
    L_Lock_1_Close_T : TP;
    L_Lock_2_Open_T : TP;
    L_Lock_2_Close_T : TP;
    L_Prev_Armed : BOOL;
    L_Auto_Lock_Req : BOOL;
    R_Trig_Gate : R_TRIG;
    R_Trig_Wicket : R_TRIG;
    R_Trig_Lock_1_O : R_TRIG;
    R_Trig_Lock_1_C : R_TRIG;
    R_Trig_Lock_2_O : R_TRIG;
    R_Trig_Lock_2_C : R_TRIG;
    fbAccessCode : FB_AccessCode_Manager;
    L_Valid_PIN : BOOL;
  END_VAR

            // Если ПЛК находится в режиме Standby (резерв), он не должен управлять выходами
IF NOT VI_IsActivePLC THEN
    RETURN;
END_IF;

IF VI_System_Mode = E_System_Operating_Mode.MODE_SAFE_STOP THEN
    VO_Gate_Open := FALSE;
    VO_Wicket_Open := FALSE;
    VO_Lock_1_Open := FALSE;
    VO_Lock_2_Open := FALSE;
    RETURN;
END_IF;

// 1. Логика автоматического закрытия замков при постановке на охрану (ТЗ 3.0)
// При переходе системы в режим "Охрана" принудительно блокируем все замки
IF VI_Armed AND NOT L_Prev_Armed THEN
    L_Auto_Lock_Req := TRUE;
END_IF;
L_Prev_Armed := VI_Armed;

// Детекторы фронта для команд
R_Trig_Gate(CLK := VI_Gate_Open_Req);
R_Trig_Wicket(CLK := VI_Wicket_Open_Req);
R_Trig_Lock_1_O(CLK := VI_Lock_1_Open_Req);
R_Trig_Lock_1_C(CLK := VI_Lock_1_Close_Req OR L_Auto_Lock_Req);
R_Trig_Lock_2_O(CLK := VI_Lock_2_Open_Req);
R_Trig_Lock_2_C(CLK := VI_Lock_2_Close_Req OR L_Auto_Lock_Req);

// Проверка PIN-кода или RFID-метки через менеджер кодов
fbAccessCode(
    VI_System_Time_MS := VI_System_Time_MS,
    VI_IsActivePLC := VI_IsActivePLC,
    VI_Code_To_Check := VI_PIN_Code,
    VI_RFID_To_Check := VI_RFID_Tag,
    VI_Access_Codes := VI_Access_Codes,
    VI_RFID_Tags := VI_RFID_Tags,
    VO_Code_Valid => L_Valid_PIN
);

// 2. Формирование импульсов управления исполнительными механизмами (Pulse Control)
// Открытие ворот и калитки требует валидного ПИН-кода или RFID-метки, если система под охраной
L_Gate_Timer(IN := R_Trig_Gate.Q AND (NOT VI_Armed OR L_Valid_PIN), PT := TO_TIME(VI_Config.gate_open_pulse_ms));
VO_Gate_Open := L_Gate_Timer.Q;

L_Wicket_Timer(IN := R_Trig_Wicket.Q AND (NOT VI_Armed OR L_Valid_PIN), PT := TO_TIME(VI_Config.wicket_open_pulse_ms));
VO_Wicket_Open := L_Wicket_Timer.Q;

L_Lock_1_Open_T(IN := R_Trig_Lock_1_O.Q AND (NOT VI_Armed OR L_Valid_PIN), PT := TO_TIME(VI_Config.lock_open_pulse_ms));
VO_Lock_1_Open := L_Lock_1_Open_T.Q;

L_Lock_1_Close_T(IN := R_Trig_Lock_1_C.Q, PT := TO_TIME(VI_Config.lock_close_pulse_ms));
VO_Lock_1_Close := L_Lock_1_Close_T.Q;

L_Lock_2_Open_T(IN := R_Trig_Lock_2_O.Q AND (NOT VI_Armed OR L_Valid_PIN), PT := TO_TIME(VI_Config.lock_open_pulse_ms));
VO_Lock_2_Open := L_Lock_2_Open_T.Q;

L_Lock_2_Close_T(IN := R_Trig_Lock_2_C.Q, PT := TO_TIME(VI_Config.lock_close_pulse_ms));
VO_Lock_2_Close := L_Lock_2_Close_T.Q;

// Сброс флага автоматического закрытия
IF L_Auto_Lock_Req THEN
    L_Auto_Lock_Req := FALSE;
END_IF;
// >>> BULK_SYNC_ANCHOR: FB_Access_Control <<<
          
END_FUNCTION_BLOCK

FUNCTION_BLOCK FB_Alarm_Compatibility_Package
  VAR_INPUT
    VI_Alarm_Legacy : ST_Alarm_Record;
  END_VAR
  VAR_OUTPUT
    VO_OK : BOOL;
    VO_Alarm_Legacy_Roundtrip : ST_Alarm_Record;
  END_VAR

            VO_OK := TRUE;
VO_Alarm_Legacy_Roundtrip := VI_Alarm_Legacy;
          
END_FUNCTION_BLOCK

FUNCTION_BLOCK FB_Alarm_Manager
  VAR_INPUT
    VI_System_Time_MS : UDINT;
    VI_IsActivePLC : BOOL;
    VI_Gas_Alarm : BOOL;
    VI_Fire_Alarm : BOOL;
    VI_Flood_Alarm : BOOL;
    VI_Security_Alarm : BOOL;
    VI_First_Fault_Active : BOOL;
    VI_First_Fault_Type : INT;
    VI_First_Fault_Source : INT;
    VI_Security_Msg : STRING(200);
    VI_Acknowledge_All : BOOL;
    VI_Mute_Siren : BOOL;
  END_VAR
  VAR_OUTPUT
    VO_Global_Critical : BOOL;
    VO_Global_Warning : BOOL;
    VO_Siren_Active : BOOL;
    VO_Active_Count : INT;
    VO_Unacked_Count : INT;
    VO_Event_Pulse : BOOL;
    VO_Event_Code : UDINT;
    VO_Event_Value : REAL;
    VO_Alarm_List : ARRAY[1..GVL_CONSTANTS.C_MAX_ALARMS] OF ST_Alarm_Record;
  END_VAR
  VAR_IN_OUT
    VI_Boiler_Errors : ARRAY[1..GVL_CONSTANTS.C_MAX_BOILERS] OF BOOL;
  END_VAR
  VAR_IN_OUT
    VIO_Next_Alarm_ID : UDINT;
  END_VAR
  VAR
    fbCompatAlarm : ARRAY[1..GVL_CONSTANTS.C_MAX_ALARMS] OF FB_Alarm_Compatibility_Package;
    L_i, L_j, L_k : INT;
    L_Target_Slot : INT;
    L_Min_Pri : INT;
    L_Pending_Alarms : ARRAY[1..10] OF ST_Alarm_Record;
    L_Pending_Count : INT := 0;
    T_Debounce_Gas : FB_System_Timer;
    T_Debounce_Fire : FB_System_Timer;
    T_Debounce_Flood : FB_System_Timer;
    T_Debounce_Security : FB_System_Timer;
    R_Trig_Gas : R_TRIG;
    R_Trig_Fire : R_TRIG;
    R_Trig_Flood : R_TRIG;
    R_Trig_Security : R_TRIG;
    R_Trig_First_Fault : R_TRIG;
    R_Trig_Boiler : ARRAY[1..GVL_CONSTANTS.C_MAX_BOILERS] OF R_TRIG;
    L_First_Fault_Source_Text : STRING(32);
    L_First_Fault_Type_Text : STRING(32);
    L_Event_Pulse_Latched : BOOL;
    L_Alarm_Compat_All_OK : BOOL;
    L_Alarm_First_Warning : STRING(255);
    L_Alarm_First_Warning_Latched : BOOL;
    L_Alarm_Shadow_Mismatch : BOOL;
    L_Alarm_Shadow_First_Mismatch : INT;
    L_Alarm_V2_Switch_Enabled : BOOL;
    L_Alarm_V2_Path_Ready : BOOL;
    L_Alarm_Using_Legacy_Fallback : BOOL;
    fbAlarmV2Core : FB_Alarm_V2_Core;
    fbHistoryV2Core : FB_History_V2_Core;
    fbBlackBoxV2Core : FB_BlackBox_V2_Core;
    L_BlackBox_V2_Snapshot_Shadow : ST_BlackBox_Snapshot_V2;
    L_History_V2_Shadow_Diff_Found : BOOL;
    L_History_V2_Shadow_First_Diff_Slot : INT;
    L_BlackBox_V2_Shadow_Diff_Found : BOOL;
    L_History_V2_Buffer_Shadow : ARRAY[1..GVL_CONSTANTS.C_MAX_HISTORY_RECORDS] OF ST_History_Event_V2;
    L_Alarm_V2_Shadow_Compare_Enabled : BOOL;
    L_Alarm_V2_Shadow_Diff_Found : BOOL;
    L_Alarm_V2_Shadow_First_Diff_Slot : INT;
    L_Alarm_V2_Event_Pulse : BOOL;
    L_Alarm_V2_Event_Code : UDINT;
    L_Alarm_V2_Event_Value : REAL;
    L_Alarm_V2_List_Shadow : ARRAY[1..GVL_CONSTANTS.C_MAX_ALARMS] OF ST_Alarm_Record;
    L_Alarm_V2_Next_ID_Shadow : UDINT;
  END_VAR

            VO_Event_Pulse := FALSE;
VO_Event_Code := 0;
VO_Event_Value := 0.0;

L_Alarm_Compat_All_OK := TRUE;
L_Alarm_First_Warning := '';
L_Alarm_First_Warning_Latched := FALSE;
L_Alarm_Shadow_Mismatch := FALSE;
L_Alarm_Shadow_First_Mismatch := 0;
L_Alarm_V2_Switch_Enabled := TRUE;
L_Alarm_V2_Path_Ready := FALSE;
L_Alarm_Using_Legacy_Fallback := TRUE;
L_Alarm_V2_Shadow_Compare_Enabled := TRUE;
L_Alarm_V2_Shadow_Diff_Found := FALSE;
L_Alarm_V2_Shadow_First_Diff_Slot := 0;
L_Alarm_V2_Event_Pulse := FALSE;
L_Alarm_V2_Event_Code := 0;
L_Alarm_V2_Event_Value := 0.0;
L_Alarm_V2_Next_ID_Shadow := VIO_Next_Alarm_ID;
L_History_V2_Shadow_Diff_Found := FALSE;
L_History_V2_Shadow_First_Diff_Slot := 0;
L_BlackBox_V2_Shadow_Diff_Found := FALSE;

// 1. Детекция новых тревог (антидребезг + передний фронт)
T_Debounce_Gas(IN := VI_Gas_Alarm, PT := T#100ms, VI_System_Time_MS := VI_System_Time_MS);
T_Debounce_Fire(IN := VI_Fire_Alarm, PT := T#100ms, VI_System_Time_MS := VI_System_Time_MS);
T_Debounce_Flood(IN := VI_Flood_Alarm, PT := T#500ms, VI_System_Time_MS := VI_System_Time_MS);
T_Debounce_Security(IN := VI_Security_Alarm, PT := T#100ms, VI_System_Time_MS := VI_System_Time_MS);

R_Trig_Gas(CLK := T_Debounce_Gas.Q);
R_Trig_Fire(CLK := T_Debounce_Fire.Q);
R_Trig_Flood(CLK := T_Debounce_Flood.Q);
R_Trig_Security(CLK := T_Debounce_Security.Q);
R_Trig_First_Fault(CLK := VI_First_Fault_Active);
FOR L_i := 1 TO GVL_CONSTANTS.C_MAX_BOILERS DO
    R_Trig_Boiler[L_i](CLK := VI_Boiler_Errors[L_i]);
END_FOR;

// 2. Добавление новых тревог в список (Кольцевой буфер)
L_Pending_Count := 0;
L_Event_Pulse_Latched := FALSE;

IF R_Trig_Gas.Q AND L_Pending_Count < 10 THEN
    L_Pending_Count := L_Pending_Count + 1;
    L_Pending_Alarms[L_Pending_Count].Timestamp_MS := VI_System_Time_MS;
    L_Pending_Alarms[L_Pending_Count].Source := 'Gas';
    L_Pending_Alarms[L_Pending_Count].Source_ID := 0;
    L_Pending_Alarms[L_Pending_Count].Message := 'Критическая концентрация газа!';
    L_Pending_Alarms[L_Pending_Count].Severity := E_ALERT_PRIORITY.ALERT_PRIORITY_CRITICAL;
    L_Pending_Alarms[L_Pending_Count].Is_Active := TRUE;
    L_Pending_Alarms[L_Pending_Count].Is_Acknowledged := FALSE;
END_IF;

IF R_Trig_Fire.Q AND L_Pending_Count < 10 THEN
    L_Pending_Count := L_Pending_Count + 1;
    L_Pending_Alarms[L_Pending_Count].Timestamp_MS := VI_System_Time_MS;
    L_Pending_Alarms[L_Pending_Count].Source := 'Fire';
    L_Pending_Alarms[L_Pending_Count].Source_ID := 0;
    L_Pending_Alarms[L_Pending_Count].Message := 'Обнаружено задымление!';
    L_Pending_Alarms[L_Pending_Count].Severity := E_ALERT_PRIORITY.ALERT_PRIORITY_CRITICAL;
    L_Pending_Alarms[L_Pending_Count].Is_Active := TRUE;
    L_Pending_Alarms[L_Pending_Count].Is_Acknowledged := FALSE;
END_IF;

IF R_Trig_Flood.Q AND L_Pending_Count < 10 THEN
    L_Pending_Count := L_Pending_Count + 1;
    L_Pending_Alarms[L_Pending_Count].Timestamp_MS := VI_System_Time_MS;
    L_Pending_Alarms[L_Pending_Count].Source := 'Flood';
    L_Pending_Alarms[L_Pending_Count].Source_ID := 0;
    L_Pending_Alarms[L_Pending_Count].Message := 'Обнаружена протечка воды!';
    L_Pending_Alarms[L_Pending_Count].Severity := E_ALERT_PRIORITY.ALERT_PRIORITY_CRITICAL;
    L_Pending_Alarms[L_Pending_Count].Is_Active := TRUE;
    L_Pending_Alarms[L_Pending_Count].Is_Acknowledged := FALSE;
END_IF;

IF R_Trig_Security.Q AND L_Pending_Count < 10 THEN
    L_Pending_Count := L_Pending_Count + 1;
    L_Pending_Alarms[L_Pending_Count].Timestamp_MS := VI_System_Time_MS;
    L_Pending_Alarms[L_Pending_Count].Source := 'Security';
    L_Pending_Alarms[L_Pending_Count].Source_ID := 0;
    L_Pending_Alarms[L_Pending_Count].Message := VI_Security_Msg;
    L_Pending_Alarms[L_Pending_Count].Severity := E_ALERT_PRIORITY.ALERT_PRIORITY_CRITICAL;
    L_Pending_Alarms[L_Pending_Count].Is_Active := TRUE;
    L_Pending_Alarms[L_Pending_Count].Is_Acknowledged := FALSE;
END_IF;

IF R_Trig_First_Fault.Q AND L_Pending_Count < 10 THEN
    L_Pending_Count := L_Pending_Count + 1;
    L_Pending_Alarms[L_Pending_Count].Timestamp_MS := VI_System_Time_MS;
    L_Pending_Alarms[L_Pending_Count].Source := 'Diagnostics';
    L_Pending_Alarms[L_Pending_Count].Source_ID := TO_BYTE(VI_First_Fault_Source);

    CASE VI_First_Fault_Type OF
        1: L_First_Fault_Type_Text := 'IO';
        2: L_First_Fault_Type_Text := 'Sensor';
        3: L_First_Fault_Type_Text := 'Comm';
        4: L_First_Fault_Type_Text := 'Subsystem';
        ELSE L_First_Fault_Type_Text := 'Unknown';
    END_CASE;

    CASE VI_First_Fault_Source OF
        1: L_First_Fault_Source_Text := 'Heating';
        2: L_First_Fault_Source_Text := 'DHW';
        3: L_First_Fault_Source_Text := 'Ventilation';
        4: L_First_Fault_Source_Text := 'Lighting';
        5: L_First_Fault_Source_Text := 'Access';
        ELSE L_First_Fault_Source_Text := 'Unknown';
    END_CASE;

    L_Pending_Alarms[L_Pending_Count].Message := CONCAT('Diagnostics root cause: ', CONCAT(L_First_Fault_Source_Text, CONCAT(' / ', L_First_Fault_Type_Text)));
    L_Pending_Alarms[L_Pending_Count].Severity := E_ALERT_PRIORITY.ALERT_PRIORITY_HIGH;
    L_Pending_Alarms[L_Pending_Count].Is_Active := TRUE;
    L_Pending_Alarms[L_Pending_Count].Is_Acknowledged := FALSE;
END_IF;

FOR L_j := 1 TO GVL_CONSTANTS.C_MAX_BOILERS DO
    IF R_Trig_Boiler[L_j].Q AND L_Pending_Count < 10 THEN
        L_Pending_Count := L_Pending_Count + 1;
        L_Pending_Alarms[L_Pending_Count].Timestamp_MS := VI_System_Time_MS;
        L_Pending_Alarms[L_Pending_Count].Source := 'Boiler';
        L_Pending_Alarms[L_Pending_Count].Source_ID := TO_BYTE(L_j);
        L_Pending_Alarms[L_Pending_Count].Message := CONCAT('Авария котла №', INT_TO_STRING(L_j));
        L_Pending_Alarms[L_Pending_Count].Severity := E_ALERT_PRIORITY.ALERT_PRIORITY_HIGH;
        L_Pending_Alarms[L_Pending_Count].Is_Active := TRUE;
        L_Pending_Alarms[L_Pending_Count].Is_Acknowledged := FALSE;
    END_IF;
END_FOR;

// Shadow comparison: execute Alarm V2 core on a separate shadow list.
// Legacy path remains authoritative; this is diagnostics only.
IF L_Alarm_V2_Shadow_Compare_Enabled THEN
    fbAlarmV2Core(
        VI_System_Time_MS := VI_System_Time_MS,
        VI_Pending_Alarms := L_Pending_Alarms,
        VIO_Alarm_List := L_Alarm_V2_List_Shadow,
        VIO_Next_Alarm_ID := L_Alarm_V2_Next_ID_Shadow,
        VO_Event_Pulse => L_Alarm_V2_Event_Pulse,
        VO_Event_Code => L_Alarm_V2_Event_Code,
        VO_Event_Value => L_Alarm_V2_Event_Value
    );
END_IF;

// Staging integration: Alarm V2 core is called behind the phase-4 switch scaffold.
// Current state: switch remains disabled, so legacy path stays authoritative.
IF L_Alarm_V2_Switch_Enabled AND L_Alarm_V2_Path_Ready THEN
    fbAlarmV2Core(
        VI_System_Time_MS := VI_System_Time_MS,
        VI_Pending_Alarms := L_Pending_Alarms,
        VIO_Alarm_List := VO_Alarm_List,
        VIO_Next_Alarm_ID := VIO_Next_Alarm_ID
    );
END_IF;

// Обработка очереди новых тревог с учетом приоритетов
FOR L_i := 1 TO L_Pending_Count DO
    fbCompatAlarm[L_i](VI_Alarm_Legacy := L_Pending_Alarms[L_i]);

    IF NOT fbCompatAlarm[L_i].VO_OK THEN
        L_Alarm_Compat_All_OK := FALSE;
    END_IF;

    IF (NOT L_Alarm_First_Warning_Latched) AND (NOT fbCompatAlarm[L_i].VO_OK) THEN
        L_Alarm_First_Warning := 'Translation issue';
        L_Alarm_First_Warning_Latched := TRUE;
    END_IF;

    IF fbCompatAlarm[L_i].VO_Alarm_Legacy_Roundtrip.ID <> L_Pending_Alarms[L_i].ID THEN
        L_Alarm_Shadow_Mismatch := TRUE;
        IF L_Alarm_Shadow_First_Mismatch = 0 THEN
            L_Alarm_Shadow_First_Mismatch := L_i;
        END_IF;
    END_IF;
    // Phase 4 scaffold: optional Alarm V2 switch point.
    // Current state: always remain on legacy behavior.
    // Future state: when Alarm V2 path is implemented and validated,
    // this block becomes the controlled branch point.
    IF L_Alarm_V2_Switch_Enabled AND L_Alarm_V2_Path_Ready THEN
        L_Alarm_Using_Legacy_Fallback := FALSE;
        // Guarded V2 pipeline is allowed by shadow validation.
        // Current runtime logic still keeps legacy action flow authoritative until next package.
    ELSE
        L_Alarm_Using_Legacy_Fallback := TRUE;
    END_IF;

    L_Target_Slot := 0;
    
    // 1. Ищем пустой слот
    FOR L_k := 1 TO GVL_CONSTANTS.C_MAX_ALARMS DO
        IF VO_Alarm_List[L_k].ID = 0 THEN
            L_Target_Slot := L_k;
            EXIT;
        END_IF;
    END_FOR;
    
    // 2. Ищем квитированную тревогу с наименьшим приоритетом
    IF L_Target_Slot = 0 THEN
        L_Min_Pri := 999;
        FOR L_k := 1 TO GVL_CONSTANTS.C_MAX_ALARMS DO
            IF VO_Alarm_List[L_k].Is_Acknowledged AND TO_INT(VO_Alarm_List[L_k].Severity) < L_Min_Pri THEN
                L_Min_Pri := TO_INT(VO_Alarm_List[L_k].Severity);
                L_Target_Slot := L_k;
            END_IF;
        END_FOR;
    END_IF;
    
    // 3. Ищем неквитированную тревогу с наименьшим приоритетом (если он ниже добавляемой)
    IF L_Target_Slot = 0 THEN
        L_Min_Pri := 999;
        FOR L_k := 1 TO GVL_CONSTANTS.C_MAX_ALARMS DO
            IF TO_INT(VO_Alarm_List[L_k].Severity) < L_Min_Pri AND TO_INT(VO_Alarm_List[L_k].Severity) < TO_INT(L_Pending_Alarms[L_i].Severity) THEN
                L_Min_Pri := TO_INT(VO_Alarm_List[L_k].Severity);
                L_Target_Slot := L_k;
            END_IF;
        END_FOR;
    END_IF;
    
    IF L_Target_Slot = 0 THEN 
        // Буфер полон критических неквитированных тревог. Не затираем!
        CONTINUE; 
    END_IF;
    
    VO_Alarm_List[L_Target_Slot] := L_Pending_Alarms[L_i];
    VO_Alarm_List[L_Target_Slot].ID := VIO_Next_Alarm_ID;
    VIO_Next_Alarm_ID := VIO_Next_Alarm_ID + 1;
    IF VIO_Next_Alarm_ID = 0 THEN VIO_Next_Alarm_ID := 1; END_IF;
    IF NOT L_Event_Pulse_Latched THEN
        VO_Event_Pulse := TRUE;
        VO_Event_Code := 1203;
        VO_Event_Value := TO_REAL(VO_Alarm_List[L_Target_Slot].Severity);
        L_Event_Pulse_Latched := TRUE;
    END_IF;
END_FOR;

// Shadow comparison results: compare legacy output and V2 shadow output.
IF L_Alarm_V2_Shadow_Compare_Enabled THEN
    FOR L_i := 1 TO GVL_CONSTANTS.C_MAX_ALARMS DO
        IF (VO_Alarm_List[L_i].ID <> L_Alarm_V2_List_Shadow[L_i].ID)
           OR (VO_Alarm_List[L_i].Is_Active <> L_Alarm_V2_List_Shadow[L_i].Is_Active)
           OR (VO_Alarm_List[L_i].Is_Acknowledged <> L_Alarm_V2_List_Shadow[L_i].Is_Acknowledged)
           OR (VO_Alarm_List[L_i].Severity <> L_Alarm_V2_List_Shadow[L_i].Severity) THEN
            L_Alarm_V2_Shadow_Diff_Found := TRUE;
            IF L_Alarm_V2_Shadow_First_Diff_Slot = 0 THEN
                L_Alarm_V2_Shadow_First_Diff_Slot := L_i;
            END_IF;
        END_IF;
    END_FOR;
END_IF;

// 3. Обновление статуса существующих тревог (ушли ли они?)
FOR L_i := 1 TO GVL_CONSTANTS.C_MAX_ALARMS DO
    IF VO_Alarm_List[L_i].ID <> 0 THEN
        IF VO_Alarm_List[L_i].Source = 'Gas' THEN VO_Alarm_List[L_i].Is_Active := VI_Gas_Alarm;
        ELSIF VO_Alarm_List[L_i].Source = 'Fire' THEN VO_Alarm_List[L_i].Is_Active := VI_Fire_Alarm;
        ELSIF VO_Alarm_List[L_i].Source = 'Flood' THEN VO_Alarm_List[L_i].Is_Active := VI_Flood_Alarm;
        ELSIF VO_Alarm_List[L_i].Source = 'Security' THEN VO_Alarm_List[L_i].Is_Active := VI_Security_Alarm;
        ELSIF VO_Alarm_List[L_i].Source = 'Diagnostics' THEN VO_Alarm_List[L_i].Is_Active := VI_First_Fault_Active;
        ELSIF VO_Alarm_List[L_i].Source = 'Boiler' THEN 
            IF TO_INT(VO_Alarm_List[L_i].Source_ID) >= 1 AND TO_INT(VO_Alarm_List[L_i].Source_ID) <= GVL_CONSTANTS.C_MAX_BOILERS THEN
                VO_Alarm_List[L_i].Is_Active := VI_Boiler_Errors[TO_INT(VO_Alarm_List[L_i].Source_ID)];
            END_IF;
        END_IF;
    END_IF;
END_FOR;

// 4. Квитирование тревог
IF VI_Acknowledge_All THEN
    FOR L_i := 1 TO GVL_CONSTANTS.C_MAX_ALARMS DO
        IF VO_Alarm_List[L_i].ID <> 0 THEN
            VO_Alarm_List[L_i].Is_Acknowledged := TRUE;
        END_IF;
    END_FOR;

    IF NOT L_Event_Pulse_Latched THEN
        VO_Event_Pulse := TRUE;
        VO_Event_Code := 1201;
        VO_Event_Value := TO_REAL(VO_Unacked_Count);
        L_Event_Pulse_Latched := TRUE;
    END_IF;
END_IF;

// 4.5 Автоквитирование некритичных тревог, если они больше не активны
FOR L_i := 1 TO GVL_CONSTANTS.C_MAX_ALARMS DO
    IF VO_Alarm_List[L_i].ID <> 0 AND NOT VO_Alarm_List[L_i].Is_Active AND NOT VO_Alarm_List[L_i].Is_Acknowledged THEN
        IF VO_Alarm_List[L_i].Severity <> E_ALERT_PRIORITY.ALERT_PRIORITY_CRITICAL THEN
            VO_Alarm_List[L_i].Is_Acknowledged := TRUE;
        END_IF;
    END_IF;
END_FOR;

// 5. Очистка списка (удаление неактивных И квитированных тревог)
// В кольцевом буфере мы просто помечаем слот как пустой (ID = 0), без сдвига массива
FOR L_i := 1 TO GVL_CONSTANTS.C_MAX_ALARMS DO
    IF VO_Alarm_List[L_i].ID <> 0 AND NOT VO_Alarm_List[L_i].Is_Active AND VO_Alarm_List[L_i].Is_Acknowledged THEN
        // Удаляем тревогу
        VO_Alarm_List[L_i].ID := 0;
        IF NOT L_Event_Pulse_Latched THEN
            VO_Event_Pulse := TRUE;
            VO_Event_Code := 1202;
            VO_Event_Value := 0.0;
            L_Event_Pulse_Latched := TRUE;
        END_IF;
    END_IF;
END_FOR;

// Shadow bridge: Alarm -> History V2 (diagnostic only)
fbHistoryV2Core(
    VI_Event_Pulse := VO_Event_Pulse,
    VI_Event_Code := VO_Event_Code,
    VI_Event_Value := VO_Event_Value,
    VI_System_Time_MS := VI_System_Time_MS,
    VIO_History_Buffer := L_History_V2_Buffer_Shadow
);

// Shadow bridge: System -> BlackBox V2 (diagnostic only)
fbBlackBoxV2Core(
    VI_System_Time_MS := VI_System_Time_MS,
    VI_System_Mode := 0,
    VI_Critical_Alarm_Active := VO_Global_Critical,
    VI_Warning_Active := VO_Global_Warning,
    VI_First_Fault_Type := TO_BYTE(VI_First_Fault_Type),
    VI_First_Fault_Source := TO_BYTE(VI_First_Fault_Source),
    VI_Gas_Alarm := VI_Gas_Alarm,
    VI_Fire_Alarm := VI_Fire_Alarm,
    VI_Flood_Alarm := VI_Flood_Alarm,
    VO_Snapshot => L_BlackBox_V2_Snapshot_Shadow
);

// Shadow validation: History V2 / BlackBox V2
IF VO_Event_Pulse THEN
    IF (L_History_V2_Buffer_Shadow[1].Event_Code <> VO_Event_Code)
       OR (ABS(L_History_V2_Buffer_Shadow[1].Event_Value - VO_Event_Value) > 0.0001) THEN
        L_History_V2_Shadow_Diff_Found := TRUE;
        IF L_History_V2_Shadow_First_Diff_Slot = 0 THEN
            L_History_V2_Shadow_First_Diff_Slot := 1;
        END_IF;
    END_IF;
END_IF;

IF (L_BlackBox_V2_Snapshot_Shadow.Gas_Alarm <> VI_Gas_Alarm)
   OR (L_BlackBox_V2_Snapshot_Shadow.Fire_Alarm <> VI_Fire_Alarm)
   OR (L_BlackBox_V2_Snapshot_Shadow.Flood_Alarm <> VI_Flood_Alarm)
   OR (L_BlackBox_V2_Snapshot_Shadow.First_Fault_Type <> TO_BYTE(VI_First_Fault_Type))
   OR (L_BlackBox_V2_Snapshot_Shadow.First_Fault_Source <> TO_BYTE(VI_First_Fault_Source)) THEN
    L_BlackBox_V2_Shadow_Diff_Found := TRUE;
END_IF;

// Guarded V2 pipeline enable:
// V2 path is allowed only when no shadow diff is present in Alarm/History/BlackBox.
IF L_Alarm_V2_Switch_Enabled THEN
    IF (NOT L_Alarm_V2_Shadow_Diff_Found)
       AND (NOT L_History_V2_Shadow_Diff_Found)
       AND (NOT L_BlackBox_V2_Shadow_Diff_Found) THEN
        L_Alarm_V2_Path_Ready := TRUE;
        L_Alarm_Using_Legacy_Fallback := FALSE;
    ELSE
        L_Alarm_V2_Path_Ready := FALSE;
        L_Alarm_Using_Legacy_Fallback := TRUE;
    END_IF;
ELSE
    L_Alarm_V2_Path_Ready := FALSE;
    L_Alarm_Using_Legacy_Fallback := TRUE;
END_IF;

// 6. Подсчет статистики и формирование глобальных флагов
VO_Global_Critical := FALSE;
VO_Global_Warning := FALSE;
VO_Siren_Active := FALSE;
VO_Active_Count := 0;
VO_Unacked_Count := 0;

FOR L_i := 1 TO GVL_CONSTANTS.C_MAX_ALARMS DO
    IF VO_Alarm_List[L_i].ID <> 0 THEN
        IF VO_Alarm_List[L_i].Is_Active THEN
            VO_Active_Count := VO_Active_Count + 1;
        END_IF;
        
        IF NOT VO_Alarm_List[L_i].Is_Acknowledged THEN
            VO_Unacked_Count := VO_Unacked_Count + 1;
            
            IF VO_Alarm_List[L_i].Severity = E_ALERT_PRIORITY.ALERT_PRIORITY_CRITICAL THEN
                VO_Global_Critical := TRUE;
                // Сирена работает только для неквитированных критических тревог, если не включен Mute
                IF NOT VI_Mute_Siren THEN
                    VO_Siren_Active := TRUE;
                END_IF;
            ELSIF VO_Alarm_List[L_i].Severity = E_ALERT_PRIORITY.ALERT_PRIORITY_HIGH THEN
                VO_Global_Warning := TRUE;
            END_IF;
        END_IF;
    END_IF;
END_FOR;
// >>> BULK_SYNC_ANCHOR: FB_Alarm_Manager <<<
          
END_FUNCTION_BLOCK

FUNCTION_BLOCK FB_Alarm_V2_Core
  VAR_INPUT
    VI_System_Time_MS : UDINT;
    VI_Pending_Alarms : ARRAY[1..10] OF ST_Alarm_Record;
  END_VAR
  VAR_OUTPUT
    VO_Event_Pulse : BOOL;
    VO_Event_Code : UDINT;
    VO_Event_Value : REAL;
  END_VAR
  VAR_IN_OUT
    VIO_Alarm_List : ARRAY[1..GVL_CONSTANTS.C_MAX_ALARMS] OF ST_Alarm_Record;
    VIO_Next_Alarm_ID : UDINT;
  END_VAR

            VO_Event_Pulse := FALSE;
VO_Event_Code := 0;
VO_Event_Value := 0.0;
          
END_FUNCTION_BLOCK

FUNCTION_BLOCK FB_Analog_Validator
  VAR_INPUT
    VI_Value : REAL;
    VI_Min_Valid : REAL;
    VI_Max_Valid : REAL;
    VI_Fallback_Mode : INT := 0;
    VI_Default_Value : REAL := 0.0;
  END_VAR
  VAR_OUTPUT
    VO_Value : REAL;
    VO_Error : BOOL;
  END_VAR
  VAR
    L_Last_Good_Value : REAL;
    L_First_Valid : BOOL := FALSE;
  END_VAR

            IF VI_Value >= VI_Min_Valid AND VI_Value <= VI_Max_Valid THEN
    VO_Error := FALSE;
    VO_Value := VI_Value;
    L_Last_Good_Value := VI_Value;
    L_First_Valid := TRUE;
ELSE
    VO_Error := TRUE;
    IF VI_Fallback_Mode = 1 OR NOT L_First_Valid THEN
        VO_Value := VI_Default_Value;
    ELSE
        VO_Value := L_Last_Good_Value;
    END_IF;
END_IF;
// >>> BULK_SYNC_ANCHOR: FB_Analog_Validator <<<
          
END_FUNCTION_BLOCK

FUNCTION_BLOCK FB_Astro_Timer
  VAR_INPUT
    VI_System_Time_MS : UDINT;
    VI_Latitude : REAL := 55.75;
    VI_Longitude : REAL := 37.61;
    VI_Timezone : REAL := 3.0;
    VI_Day_Of_Year : UINT;
  END_VAR
  VAR_OUTPUT
    VO_Sunset_Time : TOD;
    VO_Sunrise_Time : TOD;
    VO_Is_Night : BOOL;
    VO_Current_TOD : TOD;
  END_VAR
  VAR
    L_Current_TOD : TOD;
    L_Pi : REAL := 3.14159265359;
    L_Rad : REAL := 3.14159265359 / 180.0;
    L_Deg : REAL := 180.0 / 3.14159265359;
    L_B : REAL;
    L_EoT : REAL;
    L_Declination : REAL;
    L_Cos_Omega : REAL;
    L_Omega : REAL;
    L_Sunrise_Local : REAL;
    L_Sunset_Local : REAL;
  END_VAR

            // >>> SYNC_TEST_MARKER_002 <<<


L_Current_TOD := GVL_STATUS.G_Current_TOD;
VO_Current_TOD := L_Current_TOD;

// Equation of Time (EoT) in minutes
L_B := 360.0 / 365.0 * TO_REAL(VI_Day_Of_Year - 81) * L_Rad;
L_EoT := 9.87 * SIN(2.0 * L_B) - 7.53 * COS(L_B) - 1.5 * SIN(L_B);

// Solar Declination in degrees
L_Declination := 23.45 * SIN(360.0 / 365.0 * TO_REAL(VI_Day_Of_Year + 284) * L_Rad);

// Hour angle
L_Cos_Omega := -TAN(VI_Latitude * L_Rad) * TAN(L_Declination * L_Rad);

IF L_Cos_Omega > 1.0 THEN
    L_Cos_Omega := 1.0; // Polar night
ELSIF L_Cos_Omega < -1.0 THEN
    L_Cos_Omega := -1.0; // Polar day
END_IF;

L_Omega := ACOS(L_Cos_Omega) * L_Deg;

// Sunrise and Sunset in local time (hours)
L_Sunrise_Local := 12.0 - (L_Omega / 15.0) - (L_EoT / 60.0) + (VI_Timezone * 15.0 - VI_Longitude) / 15.0;
L_Sunset_Local := 12.0 + (L_Omega / 15.0) - (L_EoT / 60.0) + (VI_Timezone * 15.0 - VI_Longitude) / 15.0;

// Handle bounds
IF L_Sunrise_Local < 0.0 THEN L_Sunrise_Local := L_Sunrise_Local + 24.0; END_IF;
IF L_Sunrise_Local >= 24.0 THEN L_Sunrise_Local := L_Sunrise_Local - 24.0; END_IF;
IF L_Sunset_Local < 0.0 THEN L_Sunset_Local := L_Sunset_Local + 24.0; END_IF;
IF L_Sunset_Local >= 24.0 THEN L_Sunset_Local := L_Sunset_Local - 24.0; END_IF;

// Конвертация в TOD
VO_Sunrise_Time := TO_TOD(TO_UDINT(L_Sunrise_Local * 3600000.0));
VO_Sunset_Time := TO_TOD(TO_UDINT(L_Sunset_Local * 3600000.0));

// ТЗ 15.2: Закат + 30 мин / Рассвет - 30 мин
VO_Is_Night := (L_Current_TOD > (VO_Sunset_Time + T#30m)) OR (L_Current_TOD < (VO_Sunrise_Time - T#30m));
// >>> SYNC_TEST_MARKER_FORCE <<<
// >>> BULK_SYNC_ANCHOR: FB_Astro_Timer <<<
          
END_FUNCTION_BLOCK

FUNCTION_BLOCK FB_BlackBox_Recorder
  VAR_INPUT
    VI_Current_Data : ST_BlackBox_Record;
    VI_Freeze : BOOL;
  END_VAR
  VAR_OUTPUT
    VO_Frozen : BOOL;
    VO_Records_Count : INT;
  END_VAR
  VAR
    L_Write_Index : INT := 0;
    L_Initialized : BOOL := FALSE;
  END_VAR

            IF NOT L_Initialized THEN
    L_Write_Index := GVL_Retain.G_BlackBox_LastIndex;
    IF L_Write_Index < 0 OR L_Write_Index >= GVL_CONSTANTS.C_MAX_BLACKBOX_RECORDS THEN
        L_Write_Index := 0;
        GVL_Retain.G_BlackBox_LastIndex := 0;
    END_IF;
    L_Initialized := TRUE;
END_IF;

IF VI_Freeze THEN
    GVL_Retain.G_BlackBox_Frozen := TRUE;
END_IF;

VO_Frozen := GVL_Retain.G_BlackBox_Frozen;

IF NOT GVL_Retain.G_BlackBox_Frozen THEN
    GVL_Retain.G_BlackBox_Buffer[L_Write_Index] := VI_Current_Data;
    GVL_Retain.G_BlackBox_LastIndex := L_Write_Index;
    
    L_Write_Index := L_Write_Index + 1;
    IF L_Write_Index >= GVL_CONSTANTS.C_MAX_BLACKBOX_RECORDS THEN
        L_Write_Index := 0;
    END_IF;
END_IF;

VO_Records_Count := GVL_CONSTANTS.C_MAX_BLACKBOX_RECORDS; // Размер кольцевого буфера
// >>> BULK_SYNC_ANCHOR: FB_BlackBox_Recorder <<<
          
END_FUNCTION_BLOCK

FUNCTION_BLOCK FB_BlackBox_V2_Core
  VAR_INPUT
    VI_System_Time_MS : UDINT;
    VI_System_Mode : INT;
    VI_Critical_Alarm_Active : BOOL;
    VI_Warning_Active : BOOL;
    VI_First_Fault_Type : BYTE;
    VI_First_Fault_Source : BYTE;
    VI_Gas_Alarm : BOOL;
    VI_Fire_Alarm : BOOL;
    VI_Flood_Alarm : BOOL;
  END_VAR
  VAR_OUTPUT
    VO_Snapshot : ST_BlackBox_Snapshot_V2;
  END_VAR

            VO_Snapshot.Gas_Alarm := VI_Gas_Alarm;
VO_Snapshot.Fire_Alarm := VI_Fire_Alarm;
VO_Snapshot.Flood_Alarm := VI_Flood_Alarm;
VO_Snapshot.First_Fault_Type := VI_First_Fault_Type;
VO_Snapshot.First_Fault_Source := VI_First_Fault_Source;
          
END_FUNCTION_BLOCK

FUNCTION_BLOCK FB_Blinds_V2_Staging
  VAR_INPUT
    VI_Blind_ID : INT;
    VI_Enable : BOOL;
    VI_Position_Setpoint : BYTE;
    VI_Manual_Override : BOOL;
    VI_Scenario_ID : INT;
    VI_Safety_Mode : BOOL;
    VI_Position_Actual : BYTE;
    VI_Manual_Override_Active : BOOL;
    VI_Is_Moving : BOOL;
    VI_Alarm_Active : BOOL;
  END_VAR
  VAR_OUTPUT
    VO_Command_Shadow : ST_Blinds_Command_V2;
    VO_State_Shadow : ST_Blinds_State_V2;
  END_VAR

            VO_Command_Shadow.Position_Setpoint := VI_Position_Setpoint;
VO_State_Shadow.Position_Actual := VI_Position_Actual;
          
END_FUNCTION_BLOCK

FUNCTION_BLOCK FB_Boiler_Cascade_Manager
  VAR_INPUT
    VI_Enable : BOOL;
    VI_System_Time_MS : UDINT;
    VI_Boiler_Stop : BOOL;
    VI_DHW_Heating_Demand : BOOL;
    VI_DHW_Target_Temp : REAL;
    VI_Target_Supply_Temp : REAL;
    VI_Demand_Power : REAL;
    VI_Boiler_Flame_Status : ARRAY[1..GVL_CONSTANTS.C_MAX_BOILERS] OF BOOL;
    VI_Boiler_Error_Status : ARRAY[1..GVL_CONSTANTS.C_MAX_BOILERS] OF BOOL;
    VI_Boiler_OT_Online : ARRAY[1..GVL_CONSTANTS.C_MAX_BOILERS] OF BOOL;
    VI_Boiler_Modulation : ARRAY[1..GVL_CONSTANTS.C_MAX_BOILERS] OF REAL;
  END_VAR
  VAR_OUTPUT
    VO_Boiler_Enable : ARRAY[1..GVL_CONSTANTS.C_MAX_BOILERS] OF BOOL;
    VO_Boiler_Setpoint : ARRAY[1..GVL_CONSTANTS.C_MAX_BOILERS] OF REAL;
    VO_Lead_Boiler : BYTE;
  END_VAR
  VAR
    L_i : INT;
    L_Lead_Boiler : BYTE := 1;
    L_Last_Rotation_MS : UDINT := 0;
    L_Rotation_Initialized : BOOL := FALSE;
    L_Rotation_Period_MS : UDINT := 604800000;
    L_Lead_Available : BOOL;
    L_Reserve_Available : BOOL;
    L_Reserve_Boiler : BYTE;
    L_Start_Reserve : BOOL;
    L_Target_Setpoint : REAL;
    L_Flame_Miss_Timer : ARRAY[1..GVL_CONSTANTS.C_MAX_BOILERS] OF TON;
  END_VAR

            // Сброс выходов по умолчанию
FOR L_i := 1 TO GVL_CONSTANTS.C_MAX_BOILERS DO
    VO_Boiler_Enable[L_i] := FALSE;
    VO_Boiler_Setpoint[L_i] := 0.0;
END_FOR;

// Инициализация ротации
IF NOT L_Rotation_Initialized THEN
    L_Last_Rotation_MS := VI_System_Time_MS;
    L_Rotation_Initialized := TRUE;
END_IF;

// Принудительная остановка
IF VI_Boiler_Stop THEN
    VO_Lead_Boiler := L_Lead_Boiler;
    RETURN;
END_IF;

// Ротация строго каждые 168 часов
IF (VI_System_Time_MS - L_Last_Rotation_MS) >= L_Rotation_Period_MS THEN
    IF GVL_CONSTANTS.C_MAX_BOILERS > 1 THEN
        L_Lead_Boiler := 3 - L_Lead_Boiler;
    END_IF;
    L_Last_Rotation_MS := VI_System_Time_MS;
END_IF;

L_Reserve_Boiler := SEL(L_Lead_Boiler = 1, 1, 2);

L_Lead_Available :=
    VI_Boiler_OT_Online[L_Lead_Boiler] AND
    NOT VI_Boiler_Error_Status[L_Lead_Boiler];

L_Reserve_Available :=
    (GVL_CONSTANTS.C_MAX_BOILERS > 1) AND
    VI_Boiler_OT_Online[L_Reserve_Boiler] AND
    NOT VI_Boiler_Error_Status[L_Reserve_Boiler];

// Контроль "команда есть, пламени нет" для ведущего котла
L_Flame_Miss_Timer[L_Lead_Boiler](
    IN := VI_Enable AND L_Lead_Available AND NOT VI_DHW_Heating_Demand AND NOT VI_Boiler_Flame_Status[L_Lead_Boiler],
    PT := T#120s
);

IF L_Flame_Miss_Timer[L_Lead_Boiler].Q AND L_Reserve_Available THEN
    L_Lead_Boiler := L_Reserve_Boiler;
    L_Last_Rotation_MS := VI_System_Time_MS;
    L_Lead_Available :=
        VI_Boiler_OT_Online[L_Lead_Boiler] AND
        NOT VI_Boiler_Error_Status[L_Lead_Boiler];
    L_Reserve_Boiler := SEL(L_Lead_Boiler = 1, 1, 2);
    L_Reserve_Available :=
        (GVL_CONSTANTS.C_MAX_BOILERS > 1) AND
        VI_Boiler_OT_Online[L_Reserve_Boiler] AND
        NOT VI_Boiler_Error_Status[L_Reserve_Boiler];
END_IF;

// Нет запроса тепла
IF NOT VI_Enable THEN
    VO_Lead_Boiler := L_Lead_Boiler;
    RETURN;
END_IF;

// Целевая уставка
IF VI_DHW_Heating_Demand THEN
    L_Target_Setpoint := LIMIT(20.0, VI_DHW_Target_Temp + 15.0, 85.0);
ELSE
    L_Target_Setpoint := LIMIT(20.0, VI_Target_Supply_Temp + 5.0, 80.0);
END_IF;

// Выбор ведущего по доступности
IF NOT L_Lead_Available AND L_Reserve_Available THEN
    L_Lead_Boiler := L_Reserve_Boiler;
    L_Lead_Available := TRUE;
    L_Reserve_Boiler := SEL(L_Lead_Boiler = 1, 1, 2);
    L_Reserve_Available :=
        (GVL_CONSTANTS.C_MAX_BOILERS > 1) AND
        VI_Boiler_OT_Online[L_Reserve_Boiler] AND
        NOT VI_Boiler_Error_Status[L_Reserve_Boiler];
END_IF;

// Основной котёл
IF L_Lead_Available THEN
    VO_Boiler_Enable[L_Lead_Boiler] := TRUE;
    VO_Boiler_Setpoint[L_Lead_Boiler] := L_Target_Setpoint;
END_IF;

// Резервный котёл: >80% или отказ основного
L_Start_Reserve :=
    L_Reserve_Available AND
    (
        (VI_Demand_Power > 80.0) OR
        (NOT L_Lead_Available)
    );

IF L_Start_Reserve THEN
    VO_Boiler_Enable[L_Reserve_Boiler] := TRUE;
    VO_Boiler_Setpoint[L_Reserve_Boiler] := L_Target_Setpoint;
END_IF;

VO_Lead_Boiler := L_Lead_Boiler;
          
END_FUNCTION_BLOCK

FUNCTION_BLOCK FB_Boiler_OpenTherm_Interface
  VAR_INPUT
    VI_Enable : ARRAY[1..GVL_CONSTANTS.C_MAX_BOILERS] OF BOOL;
    VI_Setpoint : ARRAY[1..GVL_CONSTANTS.C_MAX_BOILERS] OF REAL;
    VI_OT_Online : ARRAY[1..GVL_CONSTANTS.C_MAX_BOILERS] OF BOOL;
    VI_OT_Error : ARRAY[1..GVL_CONSTANTS.C_MAX_BOILERS] OF BOOL;
  END_VAR
  VAR_OUTPUT
    VO_OT_Enable : ARRAY[1..GVL_CONSTANTS.C_MAX_BOILERS] OF BOOL;
    VO_OT_Setpoint : ARRAY[1..GVL_CONSTANTS.C_MAX_BOILERS] OF REAL;
    VO_OT_Command_Valid : ARRAY[1..GVL_CONSTANTS.C_MAX_BOILERS] OF BOOL;
  END_VAR
  VAR
    L_i : INT;
  END_VAR

            FOR L_i := 1 TO GVL_CONSTANTS.C_MAX_BOILERS DO
    VO_OT_Enable[L_i] := FALSE;
    VO_OT_Setpoint[L_i] := 0.0;
    VO_OT_Command_Valid[L_i] := FALSE;

    IF VI_Enable[L_i] AND VI_OT_Online[L_i] AND NOT VI_OT_Error[L_i] THEN
        VO_OT_Enable[L_i] := TRUE;
        VO_OT_Setpoint[L_i] := LIMIT(20.0, VI_Setpoint[L_i], 80.0);
        VO_OT_Command_Valid[L_i] := TRUE;
    END_IF;
END_FOR;
          
END_FUNCTION_BLOCK

FUNCTION_BLOCK FB_CO_Detector
  VAR_INPUT
    VI_CO_PPM : REAL;
    VI_Threshold_Warning : REAL := 30.0;
    VI_Threshold_Alarm : REAL := 70.0;
  END_VAR
  VAR_OUTPUT
    VO_CO_Warning_Level : BOOL;
    VO_CO_Alarm_Level : BOOL;
  END_VAR

            VO_CO_Warning_Level := (VI_CO_PPM >= VI_Threshold_Warning);
VO_CO_Alarm_Level   := (VI_CO_PPM >= VI_Threshold_Alarm);
          
END_FUNCTION_BLOCK

FUNCTION_BLOCK FB_CRC32_Calculator
  VAR
    L_Table : ARRAY[0..255] OF DWORD;
    L_Initialized : BOOL := FALSE;
  END_VAR

            METHOD Calculate : DWORD

Calculate := 0;
END_METHOD
          
END_FUNCTION_BLOCK

FUNCTION_BLOCK FB_Calibration_Manager
  VAR_INPUT
    VI_Raw_Value : REAL;
    VI_Type : BYTE;
    VI_Calib_Record : ST_Sensor_Calibration_Record;
    VI_System_Time_MS : UDINT;
    VI_Start_Verification : BOOL;
  END_VAR
  VAR_OUTPUT
    VO_Calibrated_Value : REAL;
    VO_Verification_Active : BOOL;
    VO_Verification_Failed : BOOL;
    VO_Deviation_Percent : REAL;
  END_VAR
  VAR
    L_Verification_Timer : FB_System_Timer;
    L_Initial_Value : REAL;
  END_VAR

            // 1. Расчет калиброванного значения
CASE VI_Type OF
    1: VO_Calibrated_Value := VI_Raw_Value + VI_Calib_Record.offset;
    2, 3: VO_Calibrated_Value := (VI_Raw_Value * VI_Calib_Record.multiplier) + VI_Calib_Record.offset;
END_CASE;

// 2. Верификация через 1 час (ТЗ 9.5)
IF VI_Start_Verification AND NOT VO_Verification_Active THEN
    VO_Verification_Active := TRUE;
    L_Initial_Value := VO_Calibrated_Value;
END_IF;

L_Verification_Timer(IN := VO_Verification_Active, PT := T#1h, VI_System_Time_MS := VI_System_Time_MS);

IF L_Verification_Timer.Q THEN
    VO_Verification_Active := FALSE;
    
    // ТЗ 9.5: Отклонение ≤2.0% (норма) / >5.0% (ошибка)
    IF L_Initial_Value <> 0 THEN
        VO_Deviation_Percent := ABS(VO_Calibrated_Value - L_Initial_Value) / L_Initial_Value * 100.0;
    ELSE
        VO_Deviation_Percent := 0.0;
    END_IF;
    
    VO_Verification_Failed := (VO_Deviation_Percent > 5.0);
END_IF;
          
END_FUNCTION_BLOCK

FUNCTION_BLOCK FB_Command_Deduplication
  VAR_INPUT
    VI_Command_ID : UDINT;
    VI_Command_Type : E_Gateway_Command_Type;
    VI_Command_Value : REAL;
    VI_System_Time_MS : UDINT;
  END_VAR
  VAR_OUTPUT
    VO_Is_New_Command : BOOL;
    VO_Processed_ID : UDINT;
  END_VAR
  VAR
    L_Processed_History : ARRAY[0..GVL_CONSTANTS.C_MAX_DEDUPLICATION_HISTORY-1] OF UDINT;
    L_Processed_Times : ARRAY[0..GVL_CONSTANTS.C_MAX_DEDUPLICATION_HISTORY-1] OF UDINT;
    L_History_Index : INT := 0;
    L_i : INT;
    L_Found : BOOL;
  END_VAR

            // Check if command ID is already in history
L_Found := FALSE;
FOR L_i := 0 TO GVL_CONSTANTS.C_MAX_DEDUPLICATION_HISTORY-1 DO
    IF L_Processed_History[L_i] = VI_Command_ID AND VI_Command_ID <> 0 THEN
        // Check if the command is not too old (e.g., 1 hour = 3600000 ms)
        IF (VI_System_Time_MS - L_Processed_Times[L_i]) < 3600000 THEN
            L_Found := TRUE;
            EXIT;
        END_IF;
    END_IF;
END_FOR;

IF NOT L_Found AND VI_Command_ID <> 0 THEN
    // New command detected
    VO_Is_New_Command := TRUE;
    VO_Processed_ID := VI_Command_ID;
    
    // Add to history
    L_Processed_History[L_History_Index] := VI_Command_ID;
    L_Processed_Times[L_History_Index] := VI_System_Time_MS;
    L_History_Index := L_History_Index + 1;
    IF L_History_Index > GVL_CONSTANTS.C_MAX_DEDUPLICATION_HISTORY-1 THEN
        L_History_Index := 0;
    END_IF;
ELSE
    // Duplicate or empty command
    VO_Is_New_Command := FALSE;
    VO_Processed_ID := 0;
END_IF;
          
END_FUNCTION_BLOCK

FUNCTION_BLOCK FB_CoreKernel_Live_Observer

            
          
END_FUNCTION_BLOCK

FUNCTION_BLOCK FB_DHW_Manager
  VAR_INPUT
    VI_System_Time_MS : UDINT;
    VI_Current_TOD : TOD;
    VI_IsActivePLC : BOOL;
    VI_Temp : REAL;
    VI_Pressure : REAL;
    VI_Config : ST_DHW_Config;
    VI_Current_Day_Of_Week : UINT;
    VI_Reset_Errors : BOOL;
    VI_Emergency_Stop : BOOL;
    VI_System_Mode : E_System_Operating_Mode;
    VI_IO_Modules_Online : ARRAY[1..GVL_CONSTANTS.C_MAX_MODULES] OF BOOL;
  END_VAR
  VAR_OUTPUT
    VO_Status : ST_DHW_Status;
    VO_Heating_Pump : BOOL;
    VO_Circ_Pump : BOOL;
  END_VAR
  VAR
    fbDHWV2Staging : FB_DHW_V2_Staging;
    L_DHW_V2_Command_V2 : ST_DHW_Command_V2;
    L_DHW_V2_State_V2 : ST_DHW_State_V2;
    L_DHW_V2_Shadow_Diff_Found : BOOL;
    L_DHW_V2_Switch_Enabled : BOOL;
    L_DHW_V2_Path_Ready : BOOL;
    L_DHW_Using_Legacy_Fallback : BOOL;
    L_i : INT;
    L_Current_TOD : TOD;
    L_Legionella_Active : BOOL;
    L_Legionella_Timer : FB_System_Timer;
    L_Last_Good_Temp : REAL := 55.0;
    L_Legionella_Done_Today : BOOL;
    L_Last_Legionella_Day : UINT;
    fbTempValidator : FB_Analog_Validator;
    fbPressValidator : FB_Analog_Validator;
    L_Error_Latched : BOOL;
    L_Error_ID_Latched : WORD;
    L_Policy_Degraded : BOOL;
    L_Policy_Freeze_Protection : BOOL;
    L_Policy_Safe_Stop : BOOL;
    L_Target_Temp_Adjusted : REAL;
  END_VAR

            // >>> SYNC_TEST_MARKER_001 <<<


IF NOT VI_IsActivePLC THEN RETURN; END_IF;

L_DHW_V2_Shadow_Diff_Found := FALSE;
L_DHW_V2_Switch_Enabled := TRUE;
L_DHW_V2_Path_Ready := FALSE;
L_DHW_Using_Legacy_Fallback := TRUE;

GVL_STATE.G_DHW_IO_Fault := FALSE;
GVL_STATE.G_DHW_Sensor_Fault := FALSE;
GVL_STATE.G_DHW_Subsystem_Degraded := FALSE;

IF VI_Emergency_Stop THEN
    VO_Heating_Pump := FALSE;
    VO_Circ_Pump := FALSE;
    VO_Status.Warning := FALSE;
    VO_Status.Error := TRUE;
    VO_Status.Error_ID := TO_WORD(GVL_CONFIG.ERR_DHW_IO_OFFLINE); // временно используем общий аварийный код до детализации safety-кодов
    VO_Status.Heating_Pump_On := FALSE;
    VO_Status.Circ_Pump_On := FALSE;
    RETURN;
END_IF;

// Фиксация текущего времени
L_Current_TOD := VI_Current_TOD;

// ========================================
// DHW POLICY LAYER
// ========================================
L_Policy_Safe_Stop := (VI_System_Mode = E_System_Operating_Mode.MODE_SAFE_STOP);
L_Policy_Freeze_Protection := (VI_System_Mode = E_System_Operating_Mode.MODE_FREEZE_PROTECTION);
L_Policy_Degraded := (VI_System_Mode = E_System_Operating_Mode.MODE_DEGRADED);
L_Target_Temp_Adjusted := VI_Config.Target_Temp;
IF L_Policy_Degraded THEN
    L_Target_Temp_Adjusted := VI_Config.Target_Temp - VI_Config.Degraded_Target_Delta;
END_IF;

// ========================================
// DHW POLICY OVERRIDE
// ========================================
IF L_Policy_Safe_Stop THEN
    VO_Heating_Pump := FALSE;
    VO_Circ_Pump := FALSE;
    RETURN;
END_IF;

IF L_Policy_Freeze_Protection THEN
    VO_Heating_Pump := FALSE;
    VO_Circ_Pump := FALSE;
    RETURN;
END_IF;

// Сброс признака выполнения термодезинфекции при смене дня.
IF L_Last_Legionella_Day <> VI_Current_Day_Of_Week THEN
    L_Legionella_Done_Today := FALSE;
    L_Last_Legionella_Day := VI_Current_Day_Of_Week;
END_IF;

// Базовый сброс незащёлкнутых статусных флагов на текущий цикл.
// Критические ошибки ниже могут зафиксироваться и завершить выполнение через RETURN.
VO_Status.Warning := FALSE;
VO_Status.Error := FALSE;
VO_Status.Error_ID := 0;

// Сброс ошибок
IF VI_Reset_Errors THEN
    L_Error_Latched := FALSE;
    L_Error_ID_Latched := 0;
END_IF;

// Проверка связи с модулями ввода-вывода
FOR L_i := 1 TO GVL_CONSTANTS.C_MAX_MODULES DO
    IF NOT VI_IO_Modules_Online[L_i] THEN
        L_Error_Latched := TRUE;
        GVL_STATE.G_DHW_IO_Fault := TRUE;
        L_Error_ID_Latched := TO_WORD(GVL_CONFIG.ERR_DHW_IO_OFFLINE); // Потеря связи с модулями ввода-вывода
    END_IF;
END_FOR;

// 1. Обработка неисправностей датчиков и сервисных режимов (ТЗ 7.0)
fbTempValidator(
    VI_Value := VI_Temp,
    VI_Min_Valid := 0.0,
    VI_Max_Valid := 100.0,
    VI_Fallback_Mode := 0,
    VI_Default_Value := 55.0
);

fbPressValidator(
    VI_Value := VI_Pressure,
    VI_Min_Valid := 0.0,
    VI_Max_Valid := 10.0,
    VI_Fallback_Mode := 0
);

VO_Status.Temp := fbTempValidator.VO_Value;
VO_Status.Pressure := fbPressValidator.VO_Value;

// Сохраняем последнее достоверное значение температуры ГВС.
// Используется только для диагностики/сервиса, не для fallback-управления.
IF NOT fbTempValidator.VO_Error THEN
    L_Last_Good_Temp := VO_Status.Temp;
END_IF;

IF fbTempValidator.VO_Error THEN
    GVL_STATE.G_DHW_Sensor_Fault := TRUE;
    L_Error_Latched := TRUE;
    L_Error_ID_Latched := TO_WORD(GVL_CONFIG.ERR_DHW_TEMP_SENSOR_FAULT); // Критическая ошибка датчика температуры
ELSIF (VO_Status.Pressure < 1.0 OR VO_Status.Pressure > 4.0) AND NOT fbPressValidator.VO_Error THEN
    L_Error_Latched := TRUE;
    L_Error_ID_Latched := TO_WORD(GVL_CONFIG.ERR_DHW_PRESSURE_OUT_OF_RANGE); // Давление вне нормы
END_IF;

IF L_Error_Latched THEN
    // Критическая ошибка: переход в безопасное состояние с полной остановкой насосов.
    VO_Heating_Pump := FALSE;
    VO_Circ_Pump := FALSE;
    VO_Status.Warning := FALSE;
    VO_Status.Error := TRUE;
    VO_Status.Error_ID := L_Error_ID_Latched;
    VO_Status.Heating_Pump_On := FALSE;
    VO_Status.Circ_Pump_On := FALSE;
    RETURN;
END_IF;

// Ошибка датчика давления не останавливает ГВС,
// но переводит подсистему в режим предупреждения (degraded mode).
IF fbPressValidator.VO_Error THEN
    GVL_STATE.G_DHW_Sensor_Fault := TRUE;
    GVL_STATE.G_DHW_Subsystem_Degraded := TRUE;
    VO_Status.Warning := TRUE;
    VO_Status.Error := FALSE;
    VO_Status.Error_ID := TO_WORD(GVL_CONFIG.ERR_DHW_PRESSURE_SENSOR_FAULT);
END_IF;

// 2. Логика поддержания температуры воды в бойлере (Нагрев)
// На этом этапе FB уже выполняется только на активном ПЛК.
    
// Термическая дезинфекция (Легионелла)
IF VI_Config.Anti_Legionella_Enabled
   AND (VI_Current_Day_Of_Week = VI_Config.Anti_Legionella_Day)
   AND (L_Current_TOD >= TOD#02:00)
   AND (L_Current_TOD <= TOD#04:00)
   AND NOT L_Legionella_Done_Today THEN
    L_Legionella_Active := TRUE;
ELSE
    L_Legionella_Active := FALSE;
END_IF;

L_Legionella_Timer(IN := L_Legionella_Active AND VO_Status.Temp >= 70.0, PT := T#30m, VI_System_Time_MS := VI_System_Time_MS);
IF L_Legionella_Timer.Q THEN
    L_Legionella_Active := FALSE; // Дезинфекция завершена
    L_Legionella_Done_Today := TRUE; // Повторно в те же сутки не запускать
END_IF;

// Двухпозиционное регулирование с гистерезисом
IF L_Legionella_Active THEN
    IF VO_Status.Temp < 70.0 THEN
        VO_Heating_Pump := TRUE;
    ELSIF VO_Status.Temp > 72.0 THEN
        VO_Heating_Pump := FALSE;
    END_IF;
ELSE
    IF VO_Status.Temp < (L_Target_Temp_Adjusted - VI_Config.Hysteresis) THEN
        VO_Heating_Pump := TRUE;
    ELSIF VO_Status.Temp > (L_Target_Temp_Adjusted + VI_Config.Hysteresis) THEN
        VO_Heating_Pump := FALSE;
    END_IF;
END_IF;

// 3. Управление циркуляционным насосом ГВС по расписанию
// Рециркуляция обеспечивает мгновенное наличие горячей воды у потребителя
VO_Circ_Pump := SEL(VI_Config.Circulation_Schedule_Enabled AND NOT (VI_Config.Night_Mode_Enabled AND (L_Current_TOD < VI_Config.Circulation_Start OR L_Current_TOD > VI_Config.Circulation_End)), FALSE, TRUE);

// Формирование статусных данных для визуализации.
// К этому моменту статус уже консистентен:
// - Error = критическая ошибка с остановкой ГВС
// - Warning = деградация без остановки
VO_Status.Heating_Pump_On := VO_Heating_Pump;
VO_Status.Circ_Pump_On := VO_Circ_Pump;

// ========================================
// DHW V2 staging execution
// ========================================
fbDHWV2Staging(
    VI_Tank_ID := 1,
    VI_Enable := TRUE,
    VI_Target_Temp := VI_Config.Target_Temp,
    VI_Pump_Enable := VO_Heating_Pump,
    VI_Heating_Priority := FALSE,

    VI_Is_Active := TRUE,
    VI_Tank_Temp := VO_Status.Temp,
    VI_Supply_Temp := VO_Status.Temp,
    VI_Return_Temp := VO_Status.Temp,
    VI_Pump_Actual := VO_Heating_Pump,
    VI_Alarm_Active := VO_Status.Error,

    VO_Command_Shadow => L_DHW_V2_Command_V2,
    VO_State_Shadow => L_DHW_V2_State_V2
);

// ========================================
// DHW V2 staging validation
// ========================================
IF VO_Heating_Pump <> (L_DHW_V2_Command_V2.Pump_Enable > 0.5) THEN
    L_DHW_V2_Shadow_Diff_Found := TRUE;
END_IF;
IF ABS(VO_Status.Temp - L_DHW_V2_State_V2.Tank_Temp) > 0.1 THEN
    L_DHW_V2_Shadow_Diff_Found := TRUE;
END_IF;
IF ABS(VO_Status.Pressure - L_DHW_V2_State_V2.Supply_Temp) > 0.1 THEN
    L_DHW_V2_Shadow_Diff_Found := TRUE;
END_IF;

// Guarded DHW V2 enable
IF L_DHW_V2_Switch_Enabled THEN
    IF NOT L_DHW_V2_Shadow_Diff_Found THEN
        L_DHW_V2_Path_Ready := TRUE;
        L_DHW_Using_Legacy_Fallback := FALSE;
    ELSE
        L_DHW_V2_Path_Ready := FALSE;
        L_DHW_Using_Legacy_Fallback := TRUE;
    END_IF;
ELSE
    L_DHW_V2_Path_Ready := FALSE;
    L_DHW_Using_Legacy_Fallback := TRUE;
END_IF;

// >>> BULK_SYNC_ANCHOR: FB_DHW_Manager <<<
          
END_FUNCTION_BLOCK

FUNCTION_BLOCK FB_DHW_V2_Staging
  VAR_INPUT
    VI_Tank_ID : INT;
    VI_Enable : BOOL;
    VI_Target_Temp : REAL;
    VI_Pump_Enable : BOOL;
    VI_Heating_Priority : BOOL;
    VI_Is_Active : BOOL;
    VI_Tank_Temp : REAL;
    VI_Supply_Temp : REAL;
    VI_Return_Temp : REAL;
    VI_Pump_Actual : BOOL;
    VI_Alarm_Active : BOOL;
  END_VAR
  VAR_OUTPUT
    VO_Command_Shadow : ST_DHW_Command_V2;
    VO_State_Shadow : ST_DHW_State_V2;
  END_VAR

            IF VI_Pump_Enable THEN
    VO_Command_Shadow.Pump_Enable := 1.0;
ELSE
    VO_Command_Shadow.Pump_Enable := 0.0;
END_IF;

VO_State_Shadow.Tank_Temp := VI_Tank_Temp;
VO_State_Shadow.Supply_Temp := VI_Supply_Temp;
          
END_FUNCTION_BLOCK

FUNCTION_BLOCK FB_Debug_Logger
  VAR_INPUT
    VI_Config : ST_Debug_Logger_Config;
    VI_System_Time_MS : UDINT;
    VI_Error_Code : UDINT;
  END_VAR
  VAR_OUTPUT
    VO_Buffer : ARRAY[1..GVL_CONSTANTS.C_MAX_DEBUG_LOGS] OF ST_Debug_Log_Record;
    VO_Write_Idx : INT := 1;
    VO_Buffer_Overflow : BOOL := FALSE;
    VO_Lost_Records : UDINT := 0;
  END_VAR
  VAR_IN_OUT
    VI_Floor_Temps : ARRAY[1..GVL_CONSTANTS.C_MAX_HEATING_CIRCUITS] OF REAL;
    VI_Pump_Currents : ARRAY[1..GVL_CONSTANTS.C_MAX_MANIFOLDS] OF REAL;
  END_VAR
  VAR
    L_last_log_time : UDINT;
    L_last_temps : ARRAY[1..GVL_CONSTANTS.C_MAX_HEATING_CIRCUITS] OF REAL;
    L_last_temp_time : ARRAY[1..GVL_CONSTANTS.C_MAX_HEATING_CIRCUITS] OF UDINT;
    L_last_error : UDINT;
    L_i : INT;
    L_diff : REAL;
    L_time_diff : UDINT;
  END_VAR

            // Цикл логирования
IF VI_Config.enabled AND (SEL(VI_System_Time_MS >= L_last_log_time, VI_System_Time_MS - L_last_log_time, (4294967295 - L_last_log_time) + VI_System_Time_MS + 1)) >= VI_Config.sampling_period_ms THEN
    L_last_log_time := VI_System_Time_MS;
    
    // Логируем температуры (если изменились или по таймауту)
    FOR L_i := 1 TO GVL_CONSTANTS.C_MAX_HEATING_CIRCUITS DO
        L_diff := ABS(VI_Floor_Temps[L_i] - L_last_temps[L_i]);
        L_time_diff := (SEL(VI_System_Time_MS >= L_last_temp_time[L_i], VI_System_Time_MS - L_last_temp_time[L_i], (4294967295 - L_last_temp_time[L_i]) + VI_System_Time_MS + 1));
        
        IF (L_diff >= 0.5) OR (L_time_diff >= 3600000) THEN // Изменение на 0.5 градуса или раз в час
            L_last_temps[L_i] := VI_Floor_Temps[L_i];
            L_last_temp_time[L_i] := VI_System_Time_MS;
            
            IF VO_Buffer_Overflow THEN
                VO_Lost_Records := VO_Lost_Records + 1;
            END_IF;
            
            VO_Buffer[VO_Write_Idx].timestamp_ms := VI_System_Time_MS;
            VO_Buffer[VO_Write_Idx].level := E_Debug_Log_Level.LOG_LEVEL_VERBOSE;
            VO_Buffer[VO_Write_Idx].source_id := TO_BYTE(L_i);
            VO_Buffer[VO_Write_Idx].value_real := VI_Floor_Temps[L_i];
            VO_Buffer[VO_Write_Idx].text := 'Floor Temp Update';
            
            IF VO_Write_Idx = GVL_CONSTANTS.C_MAX_DEBUG_LOGS THEN
                VO_Buffer_Overflow := TRUE;
            END_IF;
            VO_Write_Idx := (VO_Write_Idx MOD GVL_CONSTANTS.C_MAX_DEBUG_LOGS) + 1;
        END_IF;
    END_FOR;

    // Логируем ошибки
    IF VI_Error_Code <> 0 AND VI_Error_Code <> L_last_error THEN
        L_last_error := VI_Error_Code;
        IF VO_Buffer_Overflow THEN
            VO_Lost_Records := VO_Lost_Records + 1;
        END_IF;
        
        VO_Buffer[VO_Write_Idx].timestamp_ms := VI_System_Time_MS;
        VO_Buffer[VO_Write_Idx].level := E_Debug_Log_Level.LOG_LEVEL_MINIMAL;
        VO_Buffer[VO_Write_Idx].event_code := TO_WORD(VI_Error_Code);
        VO_Buffer[VO_Write_Idx].text := 'System Error Detected';
        
        IF VO_Write_Idx = GVL_CONSTANTS.C_MAX_DEBUG_LOGS THEN
            VO_Buffer_Overflow := TRUE;
        END_IF;
        VO_Write_Idx := (VO_Write_Idx MOD GVL_CONSTANTS.C_MAX_DEBUG_LOGS) + 1;
    ELSIF VI_Error_Code = 0 THEN
        L_last_error := 0;
    END_IF;
END_IF;
          
END_FUNCTION_BLOCK

FUNCTION_BLOCK FB_Device_Predictive_Diag
  VAR_INPUT
    VI_Current_Value : REAL;
    VI_Nominal_Value : REAL;
    VI_Is_Running : BOOL;
    VI_Reset_Stats : BOOL;
    VI_System_Time_MS : UDINT;
  END_VAR
  VAR_IN_OUT
    VIO_Health_Data : ST_Device_Health;
  END_VAR
  VAR
    L_Prev_Running : BOOL;
    L_Start_Time : UDINT;
    L_Last_Calc_Time : UDINT;
    L_Elapsed_MS : UDINT;
    L_Accumulated_MS : UDINT;
    L_Timer_Running : FB_System_Timer;
  END_VAR

            // 0. Сброс статистики
IF VI_Reset_Stats THEN
    VIO_Health_Data.Starts_Count := 0;
    VIO_Health_Data.Sample_Count := 0;
    VIO_Health_Data.Current_Sum := 0.0;
    VIO_Health_Data.Avg_Start_Current := 0.0;
    VIO_Health_Data.Health_Score := 100;
    VIO_Health_Data.Maintenance_Required := FALSE;
    VIO_Health_Data.Warning_Message := '';
    VIO_Health_Data.Last_Start_Current := 0.0;
    VIO_Health_Data.Total_Runtime_Hours := 0;
    L_Accumulated_MS := 0;
END_IF;

// 1. Счётчик пусков и замер пускового тока
IF VI_Is_Running AND NOT L_Prev_Running THEN
    VIO_Health_Data.Starts_Count := VIO_Health_Data.Starts_Count + 1;
    VIO_Health_Data.Last_Start_Current := VI_Current_Value;
    L_Start_Time := VI_System_Time_MS;
    L_Last_Calc_Time := VI_System_Time_MS;
    
    // Обновление среднего пускового тока
    VIO_Health_Data.Sample_Count := VIO_Health_Data.Sample_Count + 1;
    VIO_Health_Data.Current_Sum := VIO_Health_Data.Current_Sum + VI_Current_Value;
    VIO_Health_Data.Avg_Start_Current := VIO_Health_Data.Current_Sum / UDINT_TO_REAL(VIO_Health_Data.Sample_Count);
    
    // 2. Анализ отклонения пускового тока (п. 12.1 ТЗ)
    IF VI_Current_Value > (VI_Nominal_Value * 1.5) THEN
        VIO_Health_Data.Health_Score := TO_BYTE(LIMIT(0, TO_INT(VIO_Health_Data.Health_Score) - 5, 100));
    ELSIF VI_Current_Value > (VI_Nominal_Value * 1.2) THEN
        VIO_Health_Data.Health_Score := TO_BYTE(LIMIT(0, TO_INT(VIO_Health_Data.Health_Score) - 1, 100));
    ELSIF VI_Current_Value < (VI_Nominal_Value * 0.5) THEN
        VIO_Health_Data.Health_Score := TO_BYTE(LIMIT(0, TO_INT(VIO_Health_Data.Health_Score) - 2, 100));
    END_IF;
END_IF;

// 3. Анализ рабочего тока и наработки
IF VI_Is_Running THEN
    L_Elapsed_MS := (VI_System_Time_MS - L_Last_Calc_Time);
    L_Accumulated_MS := L_Accumulated_MS + L_Elapsed_MS;
    L_Last_Calc_Time := VI_System_Time_MS;
    
    // Обновляем наработку каждый час (3600000 мс)
    IF L_Accumulated_MS >= 3600000 THEN
        VIO_Health_Data.Total_Runtime_Hours := VIO_Health_Data.Total_Runtime_Hours + 1;
        L_Accumulated_MS := L_Accumulated_MS - 3600000;
        
        // Естественный износ: -1% здоровья каждые 1000 часов
        IF (VIO_Health_Data.Total_Runtime_Hours MOD 1000) = 0 THEN
            VIO_Health_Data.Health_Score := TO_BYTE(LIMIT(0, TO_INT(VIO_Health_Data.Health_Score) - 1, 100));
        END_IF;
        
        // Анализ рабочего тока (после пускового режима)
        IF (VI_System_Time_MS - L_Start_Time) > 10000 THEN // 10 секунд после пуска
            IF VI_Current_Value > (VI_Nominal_Value * 1.1) THEN
                // Повышенный рабочий ток - ускоренный износ (-1% в час)
                VIO_Health_Data.Health_Score := TO_BYTE(LIMIT(0, TO_INT(VIO_Health_Data.Health_Score) - 1, 100));
            END_IF;
        END_IF;
    END_IF;
END_IF;

// 4. Генерация предупреждения
IF VIO_Health_Data.Health_Score < 20 THEN
    VIO_Health_Data.Maintenance_Required := TRUE;
    VIO_Health_Data.Warning_Message := 'Критический износ: проверьте механику';
ELSIF VIO_Health_Data.Health_Score < 60 THEN
    VIO_Health_Data.Maintenance_Required := FALSE;
    VIO_Health_Data.Warning_Message := 'Предупреждение: повышенное трение';
ELSE
    VIO_Health_Data.Maintenance_Required := FALSE;
    VIO_Health_Data.Warning_Message := 'В норме';
END_IF;

L_Prev_Running := VI_Is_Running;
          
END_FUNCTION_BLOCK

FUNCTION_BLOCK FB_Emergency_Valve_Open
  VAR_INPUT
    VI_Fire_Alarm : BOOL;
    VI_Gas_Alarm : BOOL;
  END_VAR
  VAR_OUTPUT
    VO_Open_Cmd : BOOL;
  END_VAR

            // Приоритетное открытие при любой серьезной аварии
VO_Open_Cmd := VI_Fire_Alarm OR VI_Gas_Alarm;
          
END_FUNCTION_BLOCK

FUNCTION_BLOCK FB_Exhaust_Ventilation_Controller
  VAR_INPUT
    VI_Humidity : REAL;
    VI_CO2 : REAL;
    VI_Config : ST_Ventilation_Unit_Config;
  END_VAR
  VAR_OUTPUT
    VO_Fan_Speed : BYTE;
  END_VAR

            IF VI_Humidity > VI_Config.Threshold_Hum THEN
    VO_Fan_Speed := 100;
ELSIF VI_CO2 > 800.0 THEN
    VO_Fan_Speed := 70;
ELSE
    VO_Fan_Speed := 40;
END_IF;
          
END_FUNCTION_BLOCK

FUNCTION_BLOCK FB_Fault_Logger
  VAR_INPUT
    VI_Severity : E_System_Severity;
    VI_RootCause : E_System_Root_Cause;
    VI_Time_MS : UDINT;
  END_VAR
  VAR_OUTPUT
    VO_Last_Event_Text : STRING(200);
    VO_Event_Count : UINT;
    VO_Last_Index : UINT;
    VO_Event_Time_MS : ARRAY[1..16] OF UDINT;
    VO_Event_Severity : ARRAY[1..16] OF E_System_Severity;
    VO_Event_RootCause : ARRAY[1..16] OF E_System_Root_Cause;
    VO_Event_Text : ARRAY[1..16] OF STRING(200);
  END_VAR
  VAR
    L_Last_Severity : E_System_Severity;
    L_Last_RootCause : E_System_Root_Cause;
    L_Write_Index : UINT := 0;
    L_Event_Text : STRING(200);
  END_VAR

            L_Event_Text := '';

IF (VI_Severity <> L_Last_Severity) OR (VI_RootCause <> L_Last_RootCause) THEN
    CASE VI_RootCause OF
        E_System_Root_Cause.ROOT_FIRE:
            L_Event_Text := 'EVENT: FIRE DETECTED';
        E_System_Root_Cause.ROOT_GAS_LEAK:
            L_Event_Text := 'EVENT: GAS LEAK';
        E_System_Root_Cause.ROOT_CO_CRITICAL:
            L_Event_Text := 'EVENT: CO CRITICAL';
        E_System_Root_Cause.ROOT_CO_WARNING:
            L_Event_Text := 'EVENT: CO WARNING';
        E_System_Root_Cause.ROOT_WATER_LEAK:
            L_Event_Text := 'EVENT: WATER LEAK';
        E_System_Root_Cause.ROOT_SENSOR_FAULT:
            L_Event_Text := 'EVENT: SENSOR FAULT';
        E_System_Root_Cause.ROOT_IO_OFFLINE:
            L_Event_Text := 'EVENT: IO OFFLINE';
        E_System_Root_Cause.ROOT_COMM_FAULT:
            L_Event_Text := 'EVENT: COMM FAULT';
        E_System_Root_Cause.ROOT_WATCHDOG_FAULT:
            L_Event_Text := 'EVENT: WATCHDOG FAULT';
        E_System_Root_Cause.ROOT_SUBSYSTEM_FAULT:
            L_Event_Text := 'EVENT: SUBSYSTEM FAULT';
        ELSE
            L_Event_Text := 'EVENT: SYSTEM STATE CHANGE';
    END_CASE;

    L_Write_Index := L_Write_Index + 1;
    IF L_Write_Index > 16 THEN
        L_Write_Index := 1;
    END_IF;

    VO_Event_Time_MS[L_Write_Index] := VI_Time_MS;
    VO_Event_Severity[L_Write_Index] := VI_Severity;
    VO_Event_RootCause[L_Write_Index] := VI_RootCause;
    VO_Event_Text[L_Write_Index] := L_Event_Text;

    VO_Last_Index := L_Write_Index;
    VO_Last_Event_Text := L_Event_Text;

    IF VO_Event_Count < 16 THEN
        VO_Event_Count := VO_Event_Count + 1;
    END_IF;
END_IF;

L_Last_Severity := VI_Severity;
L_Last_RootCause := VI_RootCause;
// >>> BULK_SYNC_ANCHOR: FB_Fault_Logger <<<
          
END_FUNCTION_BLOCK

FUNCTION_BLOCK FB_FloorHeating_Controller
  VAR_INPUT
    VI_Current_Temp : REAL;
    VI_Config : ST_FloorHeating_Circuit_Config;
    VI_Tariff : ST_Tariff_Config;
    VI_Current_Hour : UINT;
    VI_IsActivePLC : BOOL;
    VI_System_Time_MS : UDINT;
  END_VAR
  VAR_OUTPUT
    VO_Pump_Run : BOOL;
    VO_Valve_Pos : REAL;
    VO_Valve_Bool : BOOL;
    VO_Effective_Setpoint : REAL;
  END_VAR
  VAR
    L_Is_Night : BOOL;
    L_PID : FB_PID_Controller;
    L_Last_Time : UDINT;
    L_Cycle_Time_S : REAL;
    L_PWM_Period_MS : UDINT;
    L_PWM_Duty_MS : UDINT;
    L_Current_Phase_MS : UDINT;
    L_PWM_Start_Time : UDINT;
  END_VAR

            // Вычисление времени цикла
IF L_Last_Time = 0 THEN
    L_Last_Time := VI_System_Time_MS;
    L_Cycle_Time_S := 1.0;
ELSE
    L_Cycle_Time_S := UDINT_TO_REAL((SEL(VI_System_Time_MS >= L_Last_Time, VI_System_Time_MS - L_Last_Time, (4294967295 - L_Last_Time) + VI_System_Time_MS + 1))) / 1000.0;
    L_Last_Time := VI_System_Time_MS;
END_IF;
IF L_Cycle_Time_S <= 0.0 THEN L_Cycle_Time_S := 0.01; END_IF;

// 1. Определение активного тарифа
IF VI_Tariff.Enabled THEN
    IF VI_Tariff.Night_Start_Hour > VI_Tariff.Night_End_Hour THEN
        // Переход через полночь (например, 23:00 - 07:00)
        L_Is_Night := (VI_Current_Hour >= VI_Tariff.Night_Start_Hour) OR (VI_Current_Hour < VI_Tariff.Night_End_Hour);
    ELSE
        // В пределах одного дня
        L_Is_Night := (VI_Current_Hour >= VI_Tariff.Night_Start_Hour) AND (VI_Current_Hour < VI_Tariff.Night_End_Hour);
    END_IF;
ELSE
    L_Is_Night := FALSE;
END_IF;

// 2. Расчет эффективной уставки
VO_Effective_Setpoint := VI_Config.design_temp;
IF L_Is_Night THEN
    VO_Effective_Setpoint := VO_Effective_Setpoint + VI_Tariff.Boost_Delta;
END_IF;

// 3. ПИД-регулирование
L_PID(
    VI_SetPoint := VO_Effective_Setpoint,
    VI_ProcessValue := VI_Current_Temp,
    VI_Kp := VI_Config.pid_kp,
    VI_Tn := 300.0,
    VI_Tv := 0.0,
    VI_Y_Min := 0.0,
    VI_Y_Max := 100.0,
    VI_Cycle_Time_S := L_Cycle_Time_S,
    VO_Output => VO_Valve_Pos
);

// 4. ШИМ-модуляция для термоэлектрического привода
IF VI_Config.pwm_period_s > 0 THEN
    L_PWM_Period_MS := TO_UDINT(VI_Config.pwm_period_s) * 1000;
ELSE
    L_PWM_Period_MS := 600000; // 10 минут
END_IF;

L_Current_Phase_MS := (SEL(VI_System_Time_MS >= L_PWM_Start_Time, VI_System_Time_MS - L_PWM_Start_Time, (4294967295 - L_PWM_Start_Time) + VI_System_Time_MS + 1));
IF L_Current_Phase_MS >= L_PWM_Period_MS THEN
    L_PWM_Start_Time := VI_System_Time_MS - (L_Current_Phase_MS - L_PWM_Period_MS); // Сохраняем остаток для точности
    L_Current_Phase_MS := (SEL(VI_System_Time_MS >= L_PWM_Start_Time, VI_System_Time_MS - L_PWM_Start_Time, (4294967295 - L_PWM_Start_Time) + VI_System_Time_MS + 1));
END_IF;

L_PWM_Duty_MS := TO_UDINT((VO_Valve_Pos / 100.0) * TO_REAL(L_PWM_Period_MS));

IF VI_IsActivePLC THEN
    VO_Pump_Run := (VO_Valve_Pos > 5.0);
    
    IF VO_Valve_Pos >= 100.0 THEN
        VO_Valve_Bool := TRUE;
    ELSIF VO_Valve_Pos <= 0.0 THEN
        VO_Valve_Bool := FALSE;
    ELSE
        VO_Valve_Bool := (L_Current_Phase_MS <= L_PWM_Duty_MS);
    END_IF;
ELSE
    VO_Pump_Run := FALSE;
    VO_Valve_Bool := FALSE;
END_IF;
          
END_FUNCTION_BLOCK

FUNCTION_BLOCK FB_FloorHeating_Freeze_Protection
  VAR_INPUT
    VI_Outdoor_Temp : REAL;
    VI_Threshold : REAL := 7.0;
  END_VAR
  VAR_OUTPUT
    VO_Freeze_Alert : BOOL;
    VO_Pump_Force_On : BOOL;
  END_VAR
  VAR_IN_OUT
    VI_Floor_Temps : ARRAY[1..GVL_CONSTANTS.C_MAX_HEATING_CIRCUITS] OF REAL;
  END_VAR
  VAR
    L_i : INT;
  END_VAR

            VO_Freeze_Alert := FALSE;
VO_Pump_Force_On := FALSE;

FOR L_i := 1 TO GVL_CONSTANTS.C_MAX_HEATING_CIRCUITS DO
    IF VI_Floor_Temps[L_i] < VI_Threshold THEN
        VO_Freeze_Alert := TRUE;
        VO_Pump_Force_On := TRUE;
        RETURN;
    END_IF;
END_FOR;

IF VI_Outdoor_Temp < -5.0 THEN
    VO_Pump_Force_On := TRUE;
END_IF;
          
END_FUNCTION_BLOCK

FUNCTION_BLOCK FB_FloorHeating_Overheat_Protection
  VAR_INPUT
    VI_Threshold : REAL := 45.0;
  END_VAR
  VAR_OUTPUT
    VO_Overheat_Detected : BOOL;
    VO_Locked_Circuits : ARRAY[1..GVL_CONSTANTS.C_MAX_HEATING_CIRCUITS] OF BOOL;
  END_VAR
  VAR_IN_OUT
    VI_Temps : ARRAY[1..GVL_CONSTANTS.C_MAX_HEATING_CIRCUITS] OF REAL;
  END_VAR
  VAR
    L_i : INT;
  END_VAR

            VO_Overheat_Detected := FALSE;
FOR L_i := 1 TO GVL_CONSTANTS.C_MAX_HEATING_CIRCUITS DO
    IF VI_Temps[L_i] > VI_Threshold THEN
        VO_Overheat_Detected := TRUE;
        VO_Locked_Circuits[L_i] := TRUE;
    END_IF;
END_FOR;
          
END_FUNCTION_BLOCK

FUNCTION_BLOCK FB_Gas_Methane_Detector
  VAR_INPUT
    VI_Methane_LEL : REAL;
    VI_Threshold : REAL := 20.0;
  END_VAR
  VAR_OUTPUT
    VO_Gas_Detected : BOOL;
  END_VAR

            VO_Gas_Detected := (VI_Methane_LEL >= VI_Threshold);
          
END_FUNCTION_BLOCK

FUNCTION_BLOCK FB_Gas_Smoke_Manager
  VAR_INPUT
    VI_System_Time_MS : UDINT;
    VI_IsActivePLC : BOOL;
    VI_Mute_Request : BOOL;
  END_VAR
  VAR_OUTPUT
    VO_Smoke_Detected : BOOL;
    VO_Gas_Detected : BOOL;
    VO_CO_Warning_Level : BOOL;
    VO_CO_Alarm_Level : BOOL;
    VO_Siren_Active : BOOL;
    VO_Gas_Valve_Close : BOOL;
    VO_Boiler_Stop : BOOL;
    VO_Vent_PV3_Boost : BOOL;
    VO_Supply_100_Req : BOOL;
    VO_Exhaust_100_Req : BOOL;
    VO_Supply_80_Req : BOOL;
    VO_Vent_Stop : BOOL;
    VO_Status_Msg : STRING(200);
  END_VAR
  VAR_IN_OUT
    VI_Methane_LEL : ARRAY[1..GVL_CONSTANTS.C_MAX_METHANE_SENSORS] OF REAL;
    VI_CO_PPM : ARRAY[1..GVL_CONSTANTS.C_MAX_CO_SENSORS] OF REAL;
    VI_Smoke_Sensors : ARRAY[1..GVL_CONSTANTS.C_MAX_SMOKE_SENSORS] OF BOOL;
  END_VAR
  VAR
    L_Methane_Max : REAL;
    L_CO_Max : REAL;
    L_Smoke_Count : UINT;
    L_Smoke_Active : BOOL;
    L_i : INT;
    L_CO_Timer_30ppm : FB_System_Timer;
    L_CO_Timer_70ppm : FB_System_Timer;
    L_CO_Timer_400ppm : FB_System_Timer;
    L_CO_Level_30 : BOOL;
    L_CO_Level_70 : BOOL;
    L_CO_Level_400 : BOOL;
    L_Smoke_Timer : ARRAY[1..GVL_CONSTANTS.C_MAX_SMOKE_SENSORS] OF FB_System_Timer;
  END_VAR

            IF NOT VI_IsActivePLC THEN RETURN; END_IF;

// Reset outputs
VO_Smoke_Detected := FALSE;
VO_Gas_Detected := FALSE;
VO_CO_Warning_Level := FALSE;
VO_CO_Alarm_Level := FALSE;

VO_Siren_Active := FALSE;
VO_Gas_Valve_Close := FALSE;
VO_Boiler_Stop := FALSE;
VO_Vent_PV3_Boost := FALSE;
VO_Supply_100_Req := FALSE;
VO_Exhaust_100_Req := FALSE;
VO_Supply_80_Req := FALSE;
VO_Vent_Stop := FALSE;
VO_Status_Msg := 'ОК';

// --- Methane ---
L_Methane_Max := 0.0;
FOR L_i := 1 TO GVL_CONSTANTS.C_MAX_METHANE_SENSORS DO
    IF VI_Methane_LEL[L_i] > L_Methane_Max THEN
        L_Methane_Max := VI_Methane_LEL[L_i];
    END_IF;
END_FOR;

IF L_Methane_Max >= 10.0 THEN
    VO_Vent_PV3_Boost := TRUE;
END_IF;

IF L_Methane_Max >= 20.0 THEN
    VO_Gas_Detected := TRUE;
    VO_Gas_Valve_Close := TRUE;
    VO_Boiler_Stop := TRUE;
    VO_Supply_100_Req := TRUE;
END_IF;

// --- CO ---
L_CO_Max := 0.0;
FOR L_i := 1 TO GVL_CONSTANTS.C_MAX_CO_SENSORS DO
    IF VI_CO_PPM[L_i] > L_CO_Max THEN
        L_CO_Max := VI_CO_PPM[L_i];
    END_IF;
END_FOR;

L_CO_Level_30 := (L_CO_Max >= 30.0);
L_CO_Level_70 := (L_CO_Max >= 70.0);
L_CO_Level_400 := (L_CO_Max >= 400.0);

L_CO_Timer_30ppm(IN := L_CO_Level_30, PT := T#8h, VI_System_Time_MS := VI_System_Time_MS);
L_CO_Timer_70ppm(IN := L_CO_Level_70, PT := T#1h, VI_System_Time_MS := VI_System_Time_MS);
L_CO_Timer_400ppm(IN := L_CO_Level_400, PT := T#15m, VI_System_Time_MS := VI_System_Time_MS);

IF L_CO_Timer_30ppm.Q THEN
    VO_CO_Warning_Level := TRUE;
    VO_Supply_80_Req := TRUE;
END_IF;

IF L_CO_Timer_70ppm.Q OR L_CO_Timer_400ppm.Q THEN
    VO_CO_Alarm_Level := TRUE;
    VO_Supply_80_Req := TRUE;
END_IF;

// --- Smoke ---
L_Smoke_Count := 0;
L_Smoke_Active := FALSE;

FOR L_i := 1 TO GVL_CONSTANTS.C_MAX_SMOKE_SENSORS DO
    L_Smoke_Timer[L_i](IN := VI_Smoke_Sensors[L_i], PT := T#30s, VI_System_Time_MS := VI_System_Time_MS);

    IF VI_Smoke_Sensors[L_i] THEN
        L_Smoke_Count := L_Smoke_Count + 1;
    END_IF;

    IF L_Smoke_Timer[L_i].Q OR (L_Smoke_Count >= 2) THEN
        L_Smoke_Active := TRUE;
    END_IF;
END_FOR;

IF L_Smoke_Active THEN
    VO_Smoke_Detected := TRUE;
    VO_Vent_Stop := TRUE;
    VO_Boiler_Stop := TRUE;
END_IF;

// Status
IF VO_Smoke_Detected THEN
    VO_Status_Msg := 'ПОЖАР';
ELSIF VO_Gas_Detected THEN
    VO_Status_Msg := 'УТЕЧКА ГАЗА';
ELSIF VO_CO_Alarm_Level THEN
    VO_Status_Msg := 'КРИТИЧЕСКИЙ CO';
ELSIF VO_CO_Warning_Level THEN
    VO_Status_Msg := 'ПОВЫШЕННЫЙ CO';
ELSE
    VO_Status_Msg := 'ОК';
END_IF;
// >>> BULK_SYNC_ANCHOR: FB_Gas_Smoke_Manager <<<
          
END_FUNCTION_BLOCK

FUNCTION_BLOCK FB_Gas_Valve_Controller
  VAR_INPUT
    VI_System_Time : UDINT;
    VI_IsActivePLC : BOOL;
    VI_Gas_Alarm : BOOL;
    VI_Config : ST_Gas_Valve_Configuration;
  END_VAR
  VAR_INPUT
    VI_Operator_ID : STRING(10);
    VI_Force : BOOL;
  END_VAR
  VAR_INPUT
    VI_Operator_ID : STRING(10);
    VI_Force : BOOL;
  END_VAR
  VAR_OUTPUT
    VO_Valve_Closed : BOOL;
    VO_Status_Msg : STRING(200);
  END_VAR

            // При аварии газа - немедленное закрытие
IF VI_Gas_Alarm AND VI_IsActivePLC THEN
    VO_Valve_Closed := TRUE;
    VO_Status_Msg := 'ГАЗОВЫЙ КЛАПАН ЗАКРЫТ ПО АВАРИИ';
END_IF;

METHOD OpenValve : BOOL

IF VI_IsActivePLC OR VI_Force THEN
    VO_Valve_Closed := FALSE;
    OpenValve := TRUE;
END_IF;
END_METHOD

METHOD CloseValve : BOOL

VO_Valve_Closed := TRUE;
CloseValve := TRUE;
END_METHOD

METHOD GetStatus : BYTE
GetStatus := TO_BYTE(SEL(VO_Valve_Closed, 0, 1));
END_METHOD
          
END_FUNCTION_BLOCK

FUNCTION_BLOCK FB_Gateway_Interface
  VAR_INPUT
    VI_System_Time_MS : UDINT;
    VI_Local_PLC_Role : E_PLC_ROLE;
    VI_Incoming_Command : ST_Gateway_Command;
    VI_Command_Received : BOOL;
    VI_Outdoor_Temp : REAL;
    VI_Security_Armed : BOOL;
    VI_Flood_Alarm_Active : BOOL;
    VI_Gas_Alarm_Active : BOOL;
    VI_Fire_Alarm_Active : BOOL;
    VI_Methane_Concentration : REAL;
    VI_Active_Scenario : E_SCENARIO_TYPE;
    VI_Send_2FA_Req : BOOL;
    VI_2FA_Code : STRING(6);
  END_VAR
  VAR_OUTPUT
    VO_Modbus_Registers : ARRAY[0..GVL_CONSTANTS.C_MAX_MODBUS_REGISTERS-1] OF WORD;
    VO_Lighting_Override : ARRAY[1..32] OF BYTE;
    VO_Blinds_Override : ARRAY[1..GVL_CONSTANTS.C_MAX_BLINDS] OF BYTE;
    VO_Socket_Override : ARRAY[1..GVL_CONSTANTS.C_MAX_SOCKETS] OF BOOL;
    VO_Arm_Req : BOOL;
    VO_Disarm_Req : BOOL;
    VO_PIN_Code : STRING(4);
    VO_RFID_Tag : STRING(20);
    VO_2FA_Code_In : STRING(6);
    VO_Data_Ready : BOOL;
    VO_HMI_Status_Message : STRING(200);
    VO_Telegram_Msg : STRING(200);
    VO_Send_Telegram : BOOL;
    VO_Set_Scenario_Req : BOOL;
    VO_Target_Scenario : E_SCENARIO_TYPE;
    VO_Set_Temp_Req : BOOL;
    VO_Target_Zone : INT;
    VO_Target_Temp : REAL;
    VO_Set_Vent_Req : BOOL;
    VO_Target_Vent_Speed : BYTE;
    VO_Reset_Errors_Req : BOOL;
    VO_Set_Config_Req : BOOL;
    VO_Sync_Time_Req : BOOL;
    VO_New_Time_MS : UDINT;
  END_VAR
  VAR_IN_OUT
    VI_FloorHeating_Temps : ARRAY[1..8] OF REAL;
    VI_Room_Temps : ARRAY[1..16] OF REAL;
    VI_Zone_Valve_States : ARRAY[1..8] OF BOOL;
    VI_Manifold_Pressures : ARRAY[1..GVL_CONSTANTS.C_MAX_MANIFOLDS] OF REAL;
    VI_Manifold_Pump_States : ARRAY[1..GVL_CONSTANTS.C_MAX_MANIFOLDS] OF BOOL;
    VI_Lighting_Base_Levels : ARRAY[1..32] OF BYTE;
    VI_Socket_States : ARRAY[1..GVL_CONSTANTS.C_MAX_SOCKETS] OF BOOL;
    VI_Blinds_Positions : ARRAY[1..GVL_CONSTANTS.C_MAX_BLINDS] OF BYTE;
    VI_Allowed_IPs : ARRAY[1..GVL_CONSTANTS.C_MAX_ALLOWED_IPS] OF STRING(15);
  END_VAR
  VAR
    L_last_update_time : UDINT;
    L_i : INT;
    L_j : INT;
    L_idx : INT;
    L_tmp_word : WORD;
    L_Code_UDINT : UDINT;
    L_Prev_Fire : BOOL;
    L_Prev_Gas : BOOL;
    L_Prev_Flood : BOOL;
    L_Prev_Security : BOOL;
    L_Deduplicator : FB_Command_Deduplication;
    L_CRC_Calc : FB_CRC32_Calculator;
    L_Calculated_CRC : DWORD;
    L_Command_Size : UDINT;
    L_IP_Allowed : BOOL;
    L_Process_Command : ST_Gateway_Command;
    L_Has_Command_To_Process : BOOL;
  END_VAR
  VAR
    L_Command_Buffer : ARRAY[1..GVL_CONSTANTS.C_MAX_GATEWAY_COMMANDS] OF ST_Gateway_Command;
    L_Buffer_Head : INT := 1;
    L_Buffer_Tail : INT := 1;
    L_Buffer_Count : INT := 0;
  END_VAR

            // Отправка уведомлений в Telegram (ТЗ 10.2)
VO_Send_Telegram := FALSE;
IF VI_Fire_Alarm_Active AND NOT L_Prev_Fire THEN
    VO_Telegram_Msg := 'ВНИМАНИЕ! ПОЖАРНАЯ ТРЕВОГА!';
    VO_Send_Telegram := TRUE;
END_IF;
IF VI_Gas_Alarm_Active AND NOT L_Prev_Gas THEN
    VO_Telegram_Msg := 'ВНИМАНИЕ! УТЕЧКА ГАЗА!';
    VO_Send_Telegram := TRUE;
END_IF;
IF VI_Flood_Alarm_Active AND NOT L_Prev_Flood THEN
    VO_Telegram_Msg := 'ВНИМАНИЕ! ПРОТЕЧКА ВОДЫ!';
    VO_Send_Telegram := TRUE;
END_IF;
IF VI_Security_Armed AND NOT L_Prev_Security THEN
    VO_Telegram_Msg := 'ОХРАНА ВКЛЮЧЕНА';
    VO_Send_Telegram := TRUE;
ELSIF NOT VI_Security_Armed AND L_Prev_Security THEN
    VO_Telegram_Msg := 'ОХРАНА ОТКЛЮЧЕНА';
    VO_Send_Telegram := TRUE;
END_IF;

L_Prev_Fire := VI_Fire_Alarm_Active;
L_Prev_Gas := VI_Gas_Alarm_Active;
L_Prev_Flood := VI_Flood_Alarm_Active;
L_Prev_Security := VI_Security_Armed;

// Обновление данных Modbus (раз в 1 сек)
IF (VI_System_Time_MS - L_last_update_time) >= GVL_CONSTANTS.C_MS_IN_SECOND THEN
    L_last_update_time := VI_System_Time_MS;
    
    // 0: Статус ПЛК и Аварии
    L_tmp_word := 0;
    IF VI_Local_PLC_Role = E_PLC_ROLE.ROLE_ACTIVE THEN L_tmp_word := L_tmp_word OR 1; END_IF;
    IF VI_Security_Armed THEN L_tmp_word := L_tmp_word OR 2; END_IF;
    IF VI_Flood_Alarm_Active THEN L_tmp_word := L_tmp_word OR 4; END_IF;
    IF VI_Gas_Alarm_Active THEN L_tmp_word := L_tmp_word OR 8; END_IF;
    IF VI_Fire_Alarm_Active THEN L_tmp_word := L_tmp_word OR 16; END_IF;
    VO_Modbus_Registers[0] := L_tmp_word;

    // 1-16: Температуры пола (x10)
    FOR L_i := 1 TO 8 DO
        VO_Modbus_Registers[L_i] := TO_WORD(TO_INT(VI_FloorHeating_Temps[L_i] * 10.0));
    END_FOR;

    // 17-310102: Температуры помещений (x10)
    FOR L_i := 1 TO 16 DO
        VO_Modbus_Registers[16 + L_i] := TO_WORD(TO_INT(VI_Room_Temps[L_i] * 10.0));
    END_FOR;

    // 310103: Состояние клапанов зон (битовая маска 1-16)
    L_tmp_word := 0;
    FOR L_i := 1 TO 8 DO
        IF VI_Zone_Valve_States[L_i] THEN
            L_tmp_word := L_tmp_word OR SHL(TO_WORD(1), L_i - 1);
        END_IF;
    END_FOR;
    VO_Modbus_Registers[33] := L_tmp_word;

    // 34-38: Давление в коллекторах (x100)
    FOR L_i := 1 TO GVL_CONSTANTS.C_MAX_MANIFOLDS DO
        VO_Modbus_Registers[33 + L_i] := TO_WORD(TO_INT(VI_Manifold_Pressures[L_i] * 100.0));
    END_FOR;

    // 40-55: Базовое освещение
    FOR L_i := 1 TO 32 DO
        VO_Modbus_Registers[39 + L_i] := TO_WORD(VI_Lighting_Base_Levels[L_i]);
    END_FOR;

    // 60-79: Положение штор (20 шт)
    FOR L_i := 1 TO GVL_CONSTANTS.C_MAX_BLINDS DO
        VO_Modbus_Registers[59 + L_i] := TO_WORD(VI_Blinds_Positions[L_i]);
    END_FOR;

    // 80-82: Розетки (битовая маска, 36 розеток -> 3 WORD)
    FOR L_i := 0 TO (GVL_CONSTANTS.C_MAX_SOCKETS - 1) / 16 DO
        L_tmp_word := 0;
        FOR L_j := 1 TO 16 DO
            L_idx := (L_i * 16) + L_j;
            IF L_idx <= GVL_CONSTANTS.C_MAX_SOCKETS THEN
                IF VI_Socket_States[L_idx] THEN
                    L_tmp_word := L_tmp_word OR SHL(TO_WORD(1), L_j - 1);
                END_IF;
            END_IF;
        END_FOR;
        VO_Modbus_Registers[79 + L_i] := L_tmp_word;
    END_FOR;

    // 100-102: 2FA Request and Code
    VO_Modbus_Registers[100] := SEL(VI_Send_2FA_Req, 0, 1);
    IF VI_Send_2FA_Req THEN
        L_Code_UDINT := STRING_TO_UDINT(VI_2FA_Code);
        VO_Modbus_Registers[101] := TO_WORD(L_Code_UDINT AND 16#FFFF);
        VO_Modbus_Registers[102] := TO_WORD(SHR(L_Code_UDINT, 16));
    ELSE
        VO_Modbus_Registers[101] := 0;
        VO_Modbus_Registers[102] := 0;
    END_IF;

    VO_Data_Ready := TRUE;
END_IF;

// Обработка входящих команд
VO_Arm_Req := FALSE;
VO_Disarm_Req := FALSE;
VO_Set_Scenario_Req := FALSE;
VO_Set_Temp_Req := FALSE;
VO_Set_Vent_Req := FALSE;
VO_Reset_Errors_Req := FALSE;
VO_Set_Config_Req := FALSE;
VO_Sync_Time_Req := FALSE;
L_Has_Command_To_Process := FALSE;

// 1. Прием команды и буферизация
IF VI_Command_Received THEN
    IF VI_Local_PLC_Role = E_PLC_ROLE.ROLE_ACTIVE THEN
        // Если активен, обрабатываем сразу
        L_Process_Command := VI_Incoming_Command;
        L_Has_Command_To_Process := TRUE;
    ELSE
        // Если резервный, добавляем в буфер
        IF L_Buffer_Count < GVL_CONSTANTS.C_MAX_GATEWAY_COMMANDS THEN
            L_Command_Buffer[L_Buffer_Head] := VI_Incoming_Command;
            L_Buffer_Head := L_Buffer_Head + 1;
            IF L_Buffer_Head > GVL_CONSTANTS.C_MAX_GATEWAY_COMMANDS THEN L_Buffer_Head := 1; END_IF;
            L_Buffer_Count := L_Buffer_Count + 1;
        END_IF;
    END_IF;
END_IF;

// 2. Извлечение из буфера при переходе в активный режим
IF NOT L_Has_Command_To_Process AND (VI_Local_PLC_Role = E_PLC_ROLE.ROLE_ACTIVE) AND (L_Buffer_Count > 0) THEN
    L_Process_Command := L_Command_Buffer[L_Buffer_Tail];
    L_Buffer_Tail := L_Buffer_Tail + 1;
    IF L_Buffer_Tail > GVL_CONSTANTS.C_MAX_GATEWAY_COMMANDS THEN L_Buffer_Tail := 1; END_IF;
    L_Buffer_Count := L_Buffer_Count - 1;
    L_Has_Command_To_Process := TRUE;
END_IF;

